// TIA Portal V16 export
// export: Created 2023-03-29T11:04:28.031083Z, ExportSetting WithDefaults, DisplayName Totally Integrated Automation Portal, DisplayVersion V16 Update 6, DisplayName TIA Portal Version Control Interface, DisplayVersion V16 Update 2, DisplayName TIA Portal Openness, DisplayVersion V16 Update 6, DisplayName STEP 7 Professional, DisplayVersion V16 Update 6, DisplayName STEP 7 Safety, DisplayVersion V16, DisplayName WinCC Advanced, DisplayVersion V16 Update 6
ORGANIZATION_BLOCK "OB1"   // OB1, LAD, ProgramCycle
TITLE = Głowny blok
{ S7_Optimized_Access := 'TRUE' }
AUTHOR : RTecmer
VERSION : 0.1
// stored: AutoNumber true, IsIECCheckEnabled false, SetENOAutomatically false
   VAR_INPUT
      Initial_Call : Bool;   // Initial call of this OB
      Remanence : Bool;   // =True, if remanent data are available
   END_VAR
   VAR_TEMP
      tempWatchDog_HMI : Int;
   END_VAR
   VAR_TEMP   // added for the SCL form of the ladder/FBD networks
      _w1 : Bool;
      _w2 : Bool;
   END_VAR
BEGIN

REGION Network 2: Zegart RTC
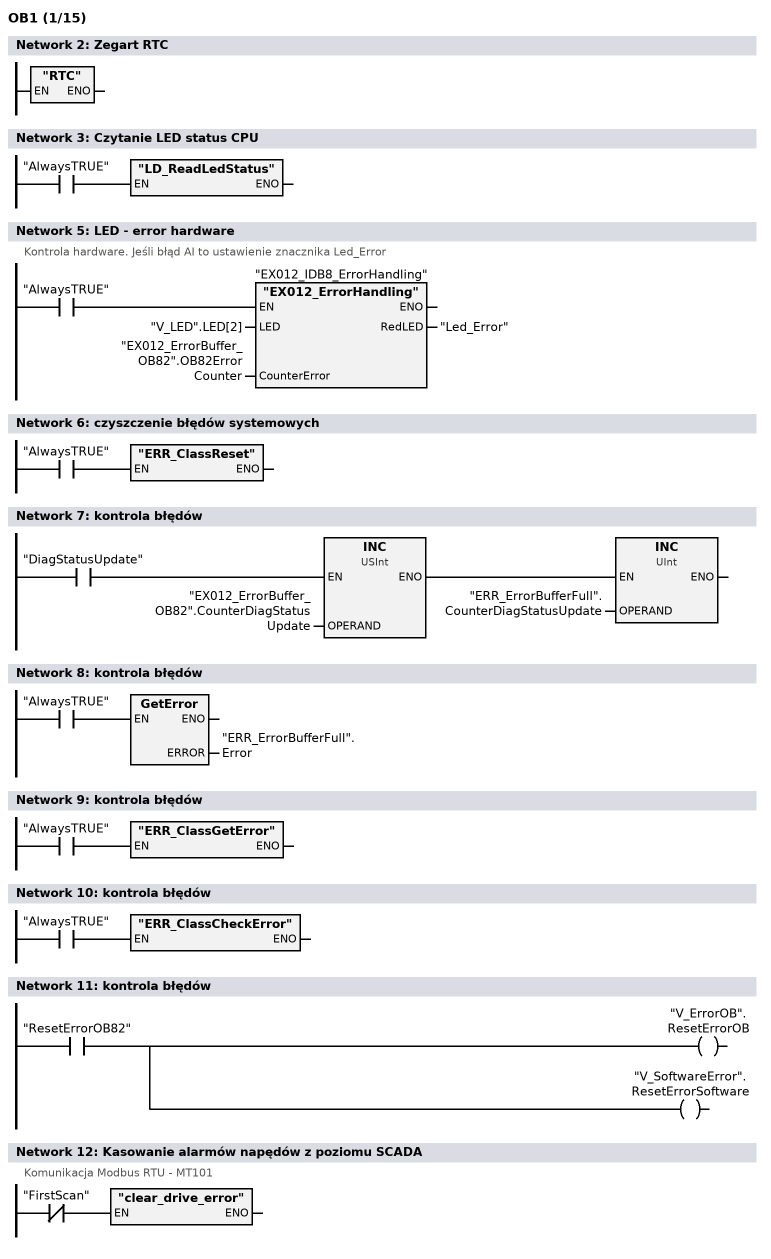
   RUNG wire#powerrail
      "RTC"()
   END_RUNG
   // the same network as SCL:
   "RTC"();
END_REGION

REGION Network 3: Czytanie LED status CPU
   RUNG wire#powerrail
      Contact( "AlwaysTRUE" )
      "LD_ReadLedStatus"()
   END_RUNG
   // the same network as SCL:
   IF "AlwaysTRUE" THEN "LD_ReadLedStatus"(); END_IF;
END_REGION

REGION Network 4 (SCL): LED kontrola RUN
   // Przekazanie  stanu LED 1 CPU
   "DB31_HMI_AreaPointer".getPLCMode := "V_LED".LED[1];
END_REGION

REGION Network 5: LED - error hardware
   // Kontrola hardware. Jeśli błąd AI to ustawienie znacznika Led_Error
   RUNG wire#powerrail
      Contact( "AlwaysTRUE" )
      "EX012_IDB8_ErrorHandling"(LED := "V_LED".LED[2], CounterError := "EX012_ErrorBuffer_OB82".OB82ErrorCounter, RedLED => "Led_Error")
   END_RUNG
   // the same network as SCL:
   IF "AlwaysTRUE" THEN
       "EX012_IDB8_ErrorHandling"(LED := "V_LED".LED[2],   // "EX012_ErrorHandling"
                               CounterError := "EX012_ErrorBuffer_OB82".OB82ErrorCounter,
                               RedLED => "Led_Error");
   END_IF;
END_REGION

REGION Network 6: czyszczenie błędów systemowych
   RUNG wire#powerrail
      Contact( "AlwaysTRUE" )
      "ERR_ClassReset"()
   END_RUNG
   // the same network as SCL:
   IF "AlwaysTRUE" THEN "ERR_ClassReset"(); END_IF;
END_REGION

REGION Network 7: kontrola błędów
   RUNG wire#powerrail
      Contact( "DiagStatusUpdate" )
      { S7_Templates := "DestType := USInt" } Inc( "EX012_ErrorBuffer_OB82".CounterDiagStatusUpdate )
      { S7_Templates := "DestType := UInt" } Inc( "ERR_ErrorBufferFull".CounterDiagStatusUpdate )
   END_RUNG
   // the same network as SCL:
   IF "DiagStatusUpdate" THEN
       "EX012_ErrorBuffer_OB82".CounterDiagStatusUpdate := "EX012_ErrorBuffer_OB82".CounterDiagStatusUpdate + 1;
       "ERR_ErrorBufferFull".CounterDiagStatusUpdate := "ERR_ErrorBufferFull".CounterDiagStatusUpdate + 1;
   END_IF;
END_REGION

REGION Network 8: kontrola błędów
   // no SCL statement known for GetError: written as a call
   IF "AlwaysTRUE" THEN GetError(error => "ERR_ErrorBufferFull".Error); END_IF;
END_REGION

REGION Network 9: kontrola błędów
   RUNG wire#powerrail
      Contact( "AlwaysTRUE" )
      "ERR_ClassGetError"()
   END_RUNG
   // the same network as SCL:
   IF "AlwaysTRUE" THEN "ERR_ClassGetError"(); END_IF;
END_REGION

REGION Network 10: kontrola błędów
   RUNG wire#powerrail
      Contact( "AlwaysTRUE" )
      "ERR_ClassCheckError"()
   END_RUNG
   // the same network as SCL:
   IF "AlwaysTRUE" THEN "ERR_ClassCheckError"(); END_IF;
END_REGION

REGION Network 11: kontrola błędów
   RUNG wire#powerrail
      Contact( "ResetErrorOB82" )
      wire#w1
      Coil( "V_ErrorOB".ResetErrorOB )
   END_RUNG
   RUNG wire#w1
      Coil( "V_SoftwareError".ResetErrorSoftware )
   END_RUNG
   // the same network as SCL:
   "V_ErrorOB".ResetErrorOB := "ResetErrorOB82";
   "V_SoftwareError".ResetErrorSoftware := "ResetErrorOB82";
END_REGION

REGION Network 12: Kasowanie alarmów napędów z poziomu SCADA
   // Komunikacja Modbus RTU - MT101
   RUNG wire#powerrail
      I_Contact( "FirstScan" )
      "clear_drive_error"()
   END_RUNG
   // the same network as SCL:
   IF NOT "FirstScan" THEN "clear_drive_error"(); END_IF;
END_REGION

REGION Network 13: Obsługa przełącznika Tryb Pracy za pośrednictwem SCADA
   // Komunikacja Modbus RTU - MT101
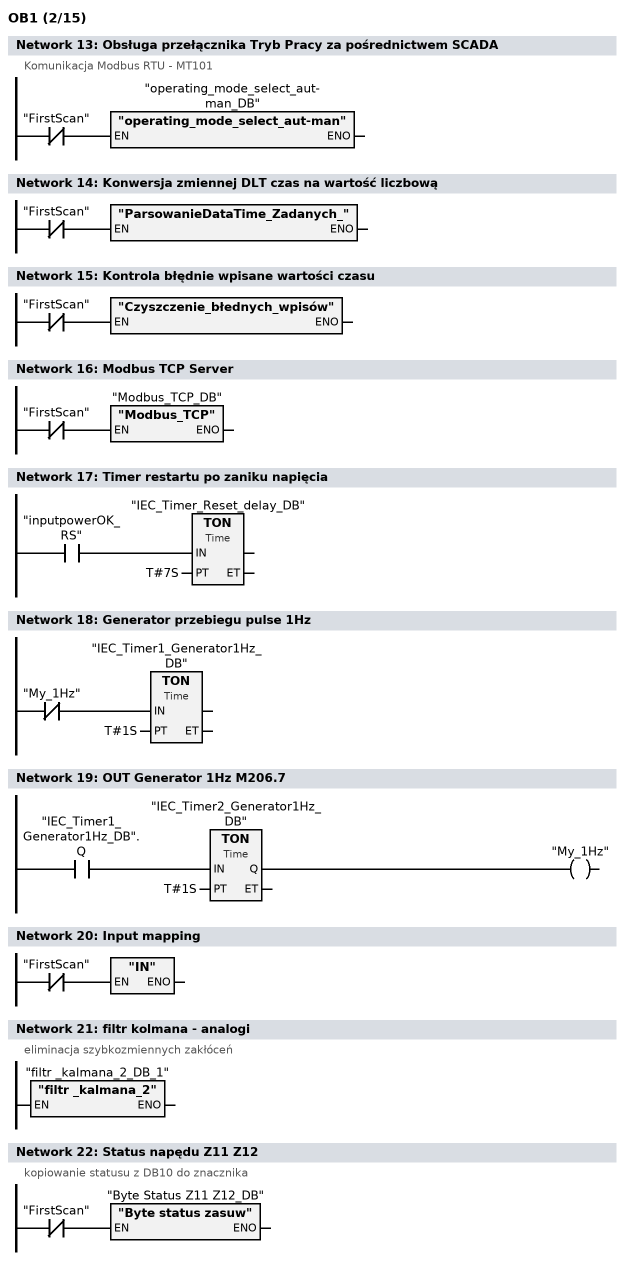
   RUNG wire#powerrail
      I_Contact( "FirstScan" )
      "operating_mode_select_aut-man_DB"()
   END_RUNG
   // the same network as SCL:
   IF NOT "FirstScan" THEN
       "operating_mode_select_aut-man_DB"();   // "operating_mode_select_aut-man"
   END_IF;
END_REGION

REGION Network 14: Konwersja zmiennej DLT czas na wartość liczbową
   RUNG wire#powerrail
      I_Contact( "FirstScan" )
      "ParsowanieDataTime_Zadanych_"()
   END_RUNG
   // the same network as SCL:
   IF NOT "FirstScan" THEN "ParsowanieDataTime_Zadanych_"(); END_IF;
END_REGION

REGION Network 15: Kontrola błędnie wpisane wartości czasu
   RUNG wire#powerrail
      I_Contact( "FirstScan" )
      "Czyszczenie_błednych_wpisów"()
   END_RUNG
   // the same network as SCL:
   IF NOT "FirstScan" THEN "Czyszczenie_błednych_wpisów"(); END_IF;
END_REGION

REGION Network 16: Modbus TCP Server
   RUNG wire#powerrail
      I_Contact( "FirstScan" )
      "Modbus_TCP_DB"()
   END_RUNG
   // the same network as SCL:
   IF NOT "FirstScan" THEN
       "Modbus_TCP_DB"();   // "Modbus_TCP"
   END_IF;
END_REGION

REGION Network 17: Timer restartu po zaniku napięcia
   RUNG wire#powerrail
      Contact( "inputpowerOK_RS" )
      { S7_Templates := "time_type := Time" } "IEC_Timer_Reset_delay_DB".TON(pt := T#7S, et =>)
   END_RUNG
   // the same network as SCL:
   "IEC_Timer_Reset_delay_DB".TON(IN := "inputpowerOK_RS", PT := T#7S);
END_REGION

REGION Network 18: Generator przebiegu pulse 1Hz
   RUNG wire#powerrail
      I_Contact( "My_1Hz" )
      { S7_Templates := "time_type := Time" } "IEC_Timer1_Generator1Hz_DB".TON(pt := T#1S, et =>)
   END_RUNG
   // the same network as SCL:
   "IEC_Timer1_Generator1Hz_DB".TON(IN := NOT "My_1Hz", PT := T#1S);
END_REGION

REGION Network 19: OUT Generator 1Hz M206.7
   RUNG wire#powerrail
      Contact( "IEC_Timer1_Generator1Hz_DB".Q )
      { S7_Templates := "time_type := Time" } "IEC_Timer2_Generator1Hz_DB".TON(pt := T#1S, et =>)
      Coil( "My_1Hz" )
   END_RUNG
   // the same network as SCL:
   "IEC_Timer2_Generator1Hz_DB".TON(IN := "IEC_Timer1_Generator1Hz_DB".Q, PT := T#1S);
   "My_1Hz" := "IEC_Timer2_Generator1Hz_DB".Q;
END_REGION

REGION Network 20: Input mapping
   RUNG wire#powerrail
      I_Contact( "FirstScan" )
      "IN"()
   END_RUNG
   // the same network as SCL:
   IF NOT "FirstScan" THEN "IN"(); END_IF;
END_REGION

REGION Network 21: filtr kolmana - analogi
   // eliminacja szybkozmiennych zakłóceń
   RUNG wire#powerrail
      "filtr _kalmana_2_DB_1"()
   END_RUNG
   // the same network as SCL:
   "filtr _kalmana_2_DB_1"();   // "filtr _kalmana_2"
END_REGION

REGION Network 22: Status napędu Z11 Z12
   // kopiowanie statusu z DB10 do znacznika
   RUNG wire#powerrail
      I_Contact( "FirstScan" )
      "Byte Status Z11 Z12_DB"()
   END_RUNG
   // the same network as SCL:
   IF NOT "FirstScan" THEN
       "Byte Status Z11 Z12_DB"();   // "Byte status zasuw"
   END_IF;
END_REGION

REGION Network 23: RTC HMI - PLC
   // Synchronizacja czasu HMI - PLC
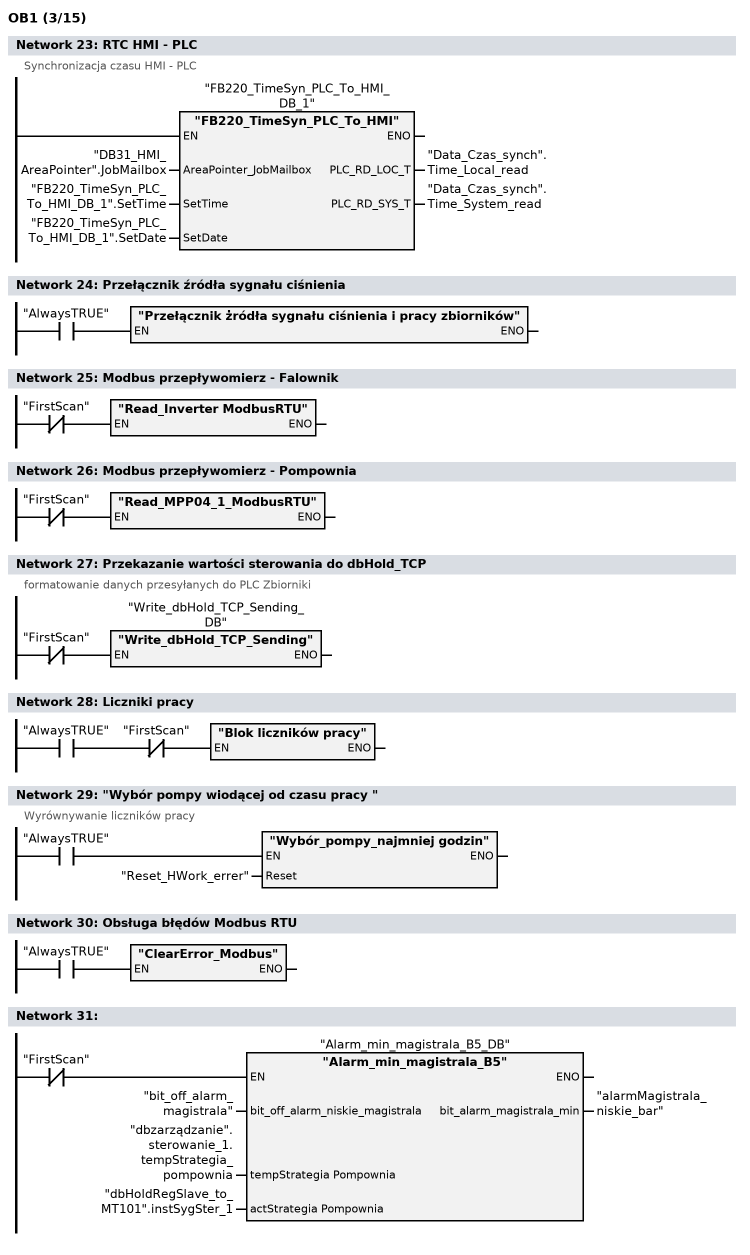
   RUNG wire#powerrail
      "FB220_TimeSyn_PLC_To_HMI_DB_1"(AreaPointer_JobMailbox := "DB31_HMI_AreaPointer".JobMailbox, SetTime := "FB220_TimeSyn_PLC_To_HMI_DB_1".SetTime, SetDate := "FB220_TimeSyn_PLC_To_HMI_DB_1".SetDate, PLC_RD_LOC_T => "Data_Czas_synch".Time_Local_read, PLC_RD_SYS_T => "Data_Czas_synch".Time_System_read)
   END_RUNG
   // the same network as SCL:
   "FB220_TimeSyn_PLC_To_HMI_DB_1"(AreaPointer_JobMailbox := "DB31_HMI_AreaPointer".JobMailbox,   // "FB220_TimeSyn_PLC_To_HMI"
                           SetTime := "FB220_TimeSyn_PLC_To_HMI_DB_1".SetTime,
                           SetDate := "FB220_TimeSyn_PLC_To_HMI_DB_1".SetDate,
                           PLC_RD_LOC_T => "Data_Czas_synch".Time_Local_read,
                           PLC_RD_SYS_T => "Data_Czas_synch".Time_System_read);
END_REGION

REGION Network 24: Przełącznik źródła sygnału ciśnienia
   RUNG wire#powerrail
      Contact( "AlwaysTRUE" )
      "Przełącznik żródła sygnału ciśnienia i pracy zbiorników"()
   END_RUNG
   // the same network as SCL:
   IF "AlwaysTRUE" THEN "Przełącznik żródła sygnału ciśnienia i pracy zbiorników"(); END_IF;
END_REGION

REGION Network 25: Modbus przepływomierz - Falownik
   RUNG wire#powerrail
      I_Contact( "FirstScan" )
      "Read_Inverter ModbusRTU"()
   END_RUNG
   // the same network as SCL:
   IF NOT "FirstScan" THEN "Read_Inverter ModbusRTU"(); END_IF;
END_REGION

REGION Network 26: Modbus przepływomierz - Pompownia
   RUNG wire#powerrail
      I_Contact( "FirstScan" )
      "Read_MPP04_1_ModbusRTU"()
   END_RUNG
   // the same network as SCL:
   IF NOT "FirstScan" THEN "Read_MPP04_1_ModbusRTU"(); END_IF;
END_REGION

REGION Network 27: Przekazanie wartości sterowania do dbHold_TCP
   // formatowanie danych przesyłanych do PLC Zbiorniki
   RUNG wire#powerrail
      I_Contact( "FirstScan" )
      "Write_dbHold_TCP_Sending_DB"()
   END_RUNG
   // the same network as SCL:
   IF NOT "FirstScan" THEN
       "Write_dbHold_TCP_Sending_DB"();   // "Write_dbHold_TCP_Sending"
   END_IF;
END_REGION

REGION Network 28: Liczniki pracy
   RUNG wire#powerrail
      Contact( "AlwaysTRUE" )
      I_Contact( "FirstScan" )
      "Blok liczników pracy"()
   END_RUNG
   // the same network as SCL:
   IF "AlwaysTRUE" AND NOT "FirstScan" THEN "Blok liczników pracy"(); END_IF;
END_REGION

REGION Network 29: "Wybór pompy wiodącej od czasu pracy "
   // Wyrównywanie liczników pracy
   RUNG wire#powerrail
      Contact( "AlwaysTRUE" )
      "Wybór_pompy_najmniej godzin"(Reset := "Reset_HWork_errer")
   END_RUNG
   // the same network as SCL:
   IF "AlwaysTRUE" THEN "Wybór_pompy_najmniej godzin"(Reset := "Reset_HWork_errer"); END_IF;
END_REGION

REGION Network 30: Obsługa błędów Modbus RTU
   RUNG wire#powerrail
      Contact( "AlwaysTRUE" )
      "ClearError_Modbus"()
   END_RUNG
   // the same network as SCL:
   IF "AlwaysTRUE" THEN "ClearError_Modbus"(); END_IF;
END_REGION

REGION Network 31
   RUNG wire#powerrail
      I_Contact( "FirstScan" )
      "Alarm_min_magistrala_B5_DB"(bit_off_alarm_niskie_magistrala := "bit_off_alarm_magistrala", "tempStrategia Pompownia" := "dbzarządzanie".sterowanie_1.tempStrategia_pompownia, "actStrategia Pompownia" := "dbHoldRegSlave_to_MT101".instSygSter_1, bit_alarm_magistrala_min => "alarmMagistrala_niskie_bar")
   END_RUNG
   // the same network as SCL:
   IF NOT "FirstScan" THEN
       "Alarm_min_magistrala_B5_DB"(bit_off_alarm_niskie_magistrala := "bit_off_alarm_magistrala",   // "Alarm_min_magistrala_B5"
                               "tempStrategia Pompownia" := "dbzarządzanie".sterowanie_1.tempStrategia_pompownia,
                               "actStrategia Pompownia" := "dbHoldRegSlave_to_MT101".instSygSter_1,
                               bit_alarm_magistrala_min => "alarmMagistrala_niskie_bar");
   END_IF;
END_REGION

REGION Network 32: Strategia sterowania zasuwami Z11
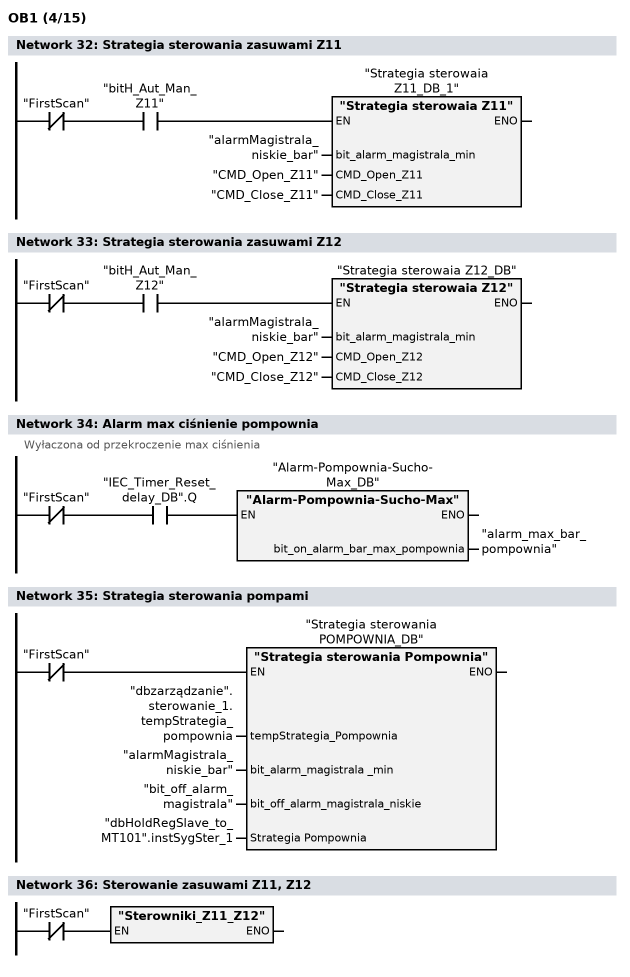
   RUNG wire#powerrail
      I_Contact( "FirstScan" )
      Contact( "bitH_Aut_Man_Z11" )
      "Strategia sterowaia Z11_DB_1"(bit_alarm_magistrala_min := "alarmMagistrala_niskie_bar", CMD_Open_Z11 := "CMD_Open_Z11", CMD_Close_Z11 := "CMD_Close_Z11")
   END_RUNG
   // the same network as SCL:
   IF NOT "FirstScan" AND "bitH_Aut_Man_Z11" THEN
       "Strategia sterowaia Z11_DB_1"(bit_alarm_magistrala_min := "alarmMagistrala_niskie_bar",   // "Strategia sterowaia Z11"
                               CMD_Open_Z11 := "CMD_Open_Z11",
                               CMD_Close_Z11 := "CMD_Close_Z11");
   END_IF;
END_REGION

REGION Network 33: Strategia sterowania zasuwami Z12
   RUNG wire#powerrail
      I_Contact( "FirstScan" )
      Contact( "bitH_Aut_Man_Z12" )
      "Strategia sterowaia Z12_DB"(bit_alarm_magistrala_min := "alarmMagistrala_niskie_bar", CMD_Open_Z12 := "CMD_Open_Z12", CMD_Close_Z12 := "CMD_Close_Z12")
   END_RUNG
   // the same network as SCL:
   IF NOT "FirstScan" AND "bitH_Aut_Man_Z12" THEN
       "Strategia sterowaia Z12_DB"(bit_alarm_magistrala_min := "alarmMagistrala_niskie_bar",   // "Strategia sterowaia Z12"
                               CMD_Open_Z12 := "CMD_Open_Z12",
                               CMD_Close_Z12 := "CMD_Close_Z12");
   END_IF;
END_REGION

REGION Network 34: Alarm max ciśnienie pompownia
   // Wyłaczona od przekroczenie max ciśnienia
   RUNG wire#powerrail
      I_Contact( "FirstScan" )
      Contact( "IEC_Timer_Reset_delay_DB".Q )
      "Alarm-Pompownia-Sucho-Max_DB"(bit_on_alarm_bar_max_pompownia => "alarm_max_bar_pompownia")
   END_RUNG
   // the same network as SCL:
   IF NOT "FirstScan" AND "IEC_Timer_Reset_delay_DB".Q THEN
       "Alarm-Pompownia-Sucho-Max_DB"(bit_on_alarm_bar_max_pompownia => "alarm_max_bar_pompownia");   // "Alarm-Pompownia-Sucho-Max"
   END_IF;
END_REGION

REGION Network 35: Strategia sterowania pompami
   RUNG wire#powerrail
      I_Contact( "FirstScan" )
      "Strategia sterowania POMPOWNIA_DB"(tempStrategia_Pompownia := "dbzarządzanie".sterowanie_1.tempStrategia_pompownia, "bit_alarm_magistrala _min" := "alarmMagistrala_niskie_bar", bit_off_alarm_magistrala_niskie := "bit_off_alarm_magistrala", "Strategia Pompownia" := "dbHoldRegSlave_to_MT101".instSygSter_1)
   END_RUNG
   // the same network as SCL:
   IF NOT "FirstScan" THEN
       "Strategia sterowania POMPOWNIA_DB"(tempStrategia_Pompownia := "dbzarządzanie".sterowanie_1.tempStrategia_pompownia,   // "Strategia sterowania Pompownia"
                               "bit_alarm_magistrala _min" := "alarmMagistrala_niskie_bar",
                               bit_off_alarm_magistrala_niskie := "bit_off_alarm_magistrala",
                               "Strategia Pompownia" := "dbHoldRegSlave_to_MT101".instSygSter_1);
   END_IF;
END_REGION

REGION Network 36: Sterowanie zasuwami Z11, Z12
   RUNG wire#powerrail
      I_Contact( "FirstScan" )
      "Sterowniki_Z11_Z12"()
   END_RUNG
   // the same network as SCL:
   IF NOT "FirstScan" THEN "Sterowniki_Z11_Z12"(); END_IF;
END_REGION

REGION Network 37: Konwerter parametrów z falownika
   // funkcja wylicza wartości pobrane z falownika protokołem Modbus RTU
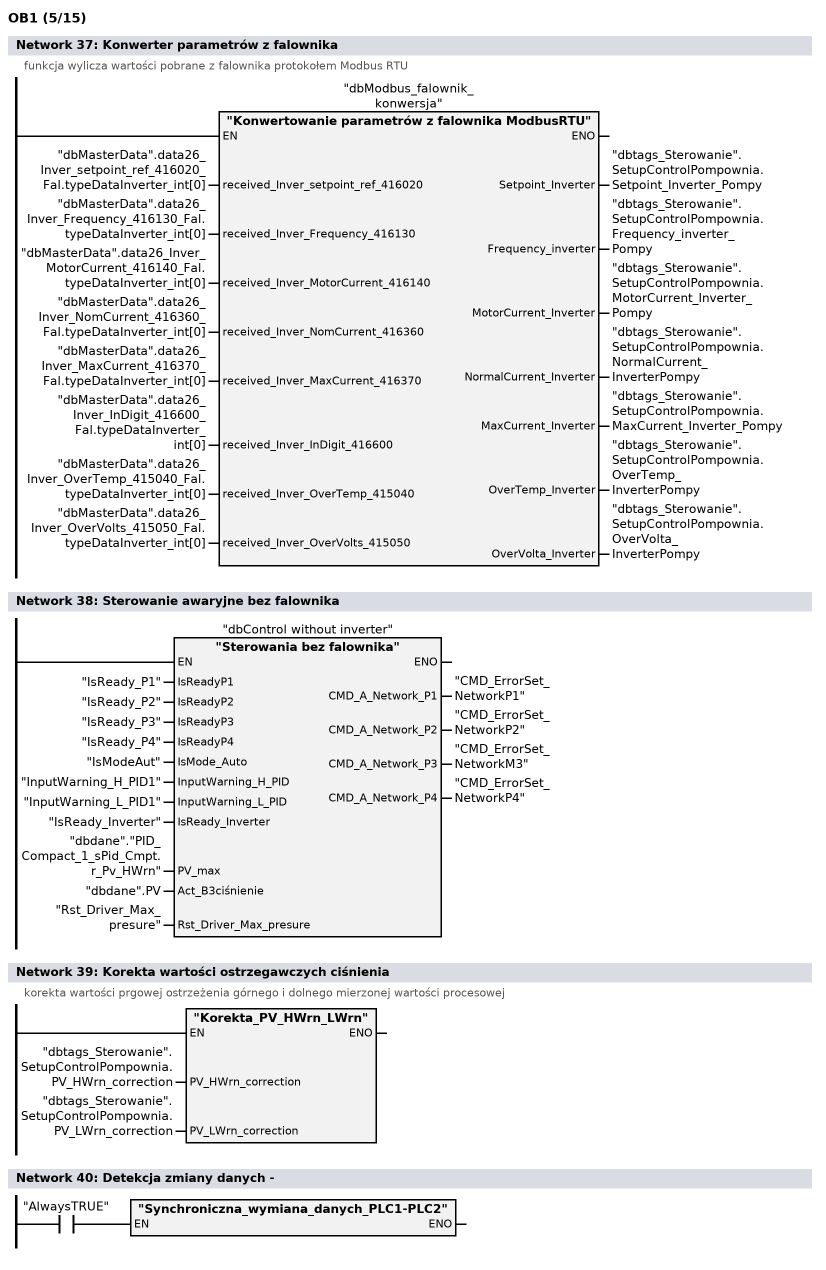
   RUNG wire#powerrail
      "dbModbus_falownik_konwersja"(received_Inver_setpoint_ref_416020 := "dbMasterData".data26_Inver_setpoint_ref_416020_Fal.typeDataInverter_int[0], received_Inver_Frequency_416130 := "dbMasterData".data26_Inver_Frequency_416130_Fal.typeDataInverter_int[0], received_Inver_MotorCurrent_416140 := "dbMasterData".data26_Inver_MotorCurrent_416140_Fal.typeDataInverter_int[0], received_Inver_NomCurrent_416360 := "dbMasterData".data26_Inver_NomCurrent_416360_Fal.typeDataInverter_int[0], received_Inver_MaxCurrent_416370 := "dbMasterData".data26_Inver_MaxCurrent_416370_Fal.typeDataInverter_int[0], received_Inver_InDigit_416600 := "dbMasterData".data26_Inver_InDigit_416600_Fal.typeDataInverter_int[0], received_Inver_OverTemp_415040 := "dbMasterData".data26_Inver_OverTemp_415040_Fal.typeDataInverter_int[0], received_Inver_OverVolts_415050 := "dbMasterData".data26_Inver_OverVolts_415050_Fal.typeDataInverter_int[0], Setpoint_Inverter => "dbtags_Sterowanie".SetupControlPompownia.Setpoint_Inverter_Pompy, Frequency_inverter => "dbtags_Sterowanie".SetupControlPompownia.Frequency_inverter_Pompy, MotorCurrent_Inverter => "dbtags_Sterowanie".SetupControlPompownia.MotorCurrent_Inverter_Pompy, NormalCurrent_Inverter => "dbtags_Sterowanie".SetupControlPompownia.NormalCurrent_InverterPompy, MaxCurrent_Inverter => "dbtags_Sterowanie".SetupControlPompownia.MaxCurrent_Inverter_Pompy, OverTemp_Inverter => "dbtags_Sterowanie".SetupControlPompownia.OverTemp_InverterPompy, OverVolta_Inverter => "dbtags_Sterowanie".SetupControlPompownia.OverVolta_InverterPompy)
   END_RUNG
   // the same network as SCL:
   "dbModbus_falownik_konwersja"(received_Inver_setpoint_ref_416020 := "dbMasterData".data26_Inver_setpoint_ref_416020_Fal.typeDataInverter_int[0],   // "Konwertowanie parametrów z falownika ModbusRTU"
                           received_Inver_Frequency_416130 := "dbMasterData".data26_Inver_Frequency_416130_Fal.typeDataInverter_int[0],
                           received_Inver_MotorCurrent_416140 := "dbMasterData".data26_Inver_MotorCurrent_416140_Fal.typeDataInverter_int[0],
                           received_Inver_NomCurrent_416360 := "dbMasterData".data26_Inver_NomCurrent_416360_Fal.typeDataInverter_int[0],
                           received_Inver_MaxCurrent_416370 := "dbMasterData".data26_Inver_MaxCurrent_416370_Fal.typeDataInverter_int[0],
                           received_Inver_InDigit_416600 := "dbMasterData".data26_Inver_InDigit_416600_Fal.typeDataInverter_int[0],
                           received_Inver_OverTemp_415040 := "dbMasterData".data26_Inver_OverTemp_415040_Fal.typeDataInverter_int[0],
                           received_Inver_OverVolts_415050 := "dbMasterData".data26_Inver_OverVolts_415050_Fal.typeDataInverter_int[0],
                           Setpoint_Inverter => "dbtags_Sterowanie".SetupControlPompownia.Setpoint_Inverter_Pompy,
                           Frequency_inverter => "dbtags_Sterowanie".SetupControlPompownia.Frequency_inverter_Pompy,
                           MotorCurrent_Inverter => "dbtags_Sterowanie".SetupControlPompownia.MotorCurrent_Inverter_Pompy,
                           NormalCurrent_Inverter => "dbtags_Sterowanie".SetupControlPompownia.NormalCurrent_InverterPompy,
                           MaxCurrent_Inverter => "dbtags_Sterowanie".SetupControlPompownia.MaxCurrent_Inverter_Pompy,
                           OverTemp_Inverter => "dbtags_Sterowanie".SetupControlPompownia.OverTemp_InverterPompy,
                           OverVolta_Inverter => "dbtags_Sterowanie".SetupControlPompownia.OverVolta_InverterPompy);
END_REGION

REGION Network 38: Sterowanie awaryjne bez falownika
   RUNG wire#powerrail
      "dbControl without inverter"(IsReadyP1 := "IsReady_P1", IsReadyP2 := "IsReady_P2", IsReadyP3 := "IsReady_P3", IsReadyP4 := "IsReady_P4", IsMode_Auto := "IsModeAut", InputWarning_H_PID := "InputWarning_H_PID1", InputWarning_L_PID := "InputWarning_L_PID1", IsReady_Inverter := "IsReady_Inverter", PV_max := "dbdane"."PID_Compact_1_sPid_Cmpt.r_Pv_HWrn", Act_B3ciśnienie := "dbdane".PV, Rst_Driver_Max_presure := "Rst_Driver_Max_presure", CMD_A_Network_P1 => "CMD_ErrorSet_NetworkP1", CMD_A_Network_P2 => "CMD_ErrorSet_NetworkP2", CMD_A_Network_P3 => "CMD_ErrorSet_NetworkM3", CMD_A_Network_P4 => "CMD_ErrorSet_NetworkP4")
   END_RUNG
   // the same network as SCL:
   "dbControl without inverter"(IsReadyP1 := "IsReady_P1",   // "Sterowania bez falownika"
                           IsReadyP2 := "IsReady_P2",
                           IsReadyP3 := "IsReady_P3",
                           IsReadyP4 := "IsReady_P4",
                           IsMode_Auto := "IsModeAut",
                           InputWarning_H_PID := "InputWarning_H_PID1",
                           InputWarning_L_PID := "InputWarning_L_PID1",
                           IsReady_Inverter := "IsReady_Inverter",
                           PV_max := "dbdane"."PID_Compact_1_sPid_Cmpt.r_Pv_HWrn",
                           Act_B3ciśnienie := "dbdane".PV,
                           Rst_Driver_Max_presure := "Rst_Driver_Max_presure",
                           CMD_A_Network_P1 => "CMD_ErrorSet_NetworkP1",
                           CMD_A_Network_P2 => "CMD_ErrorSet_NetworkP2",
                           CMD_A_Network_P3 => "CMD_ErrorSet_NetworkM3",
                           CMD_A_Network_P4 => "CMD_ErrorSet_NetworkP4");
END_REGION

REGION Network 39: Korekta wartości ostrzegawczych ciśnienia
   // korekta wartości prgowej ostrzeżenia górnego i dolnego mierzonej wartości procesowej
   RUNG wire#powerrail
      "Korekta_PV_HWrn_LWrn"(PV_HWrn_correction := "dbtags_Sterowanie".SetupControlPompownia.PV_HWrn_correction, PV_LWrn_correction := "dbtags_Sterowanie".SetupControlPompownia.PV_LWrn_correction)
   END_RUNG
   // the same network as SCL:
   "Korekta_PV_HWrn_LWrn"(PV_HWrn_correction := "dbtags_Sterowanie".SetupControlPompownia.PV_HWrn_correction,
                          PV_LWrn_correction := "dbtags_Sterowanie".SetupControlPompownia.PV_LWrn_correction);
END_REGION

REGION Network 40: Detekcja zmiany danych -
   RUNG wire#powerrail
      Contact( "AlwaysTRUE" )
      "Synchroniczna_wymiana_danych_PLC1-PLC2"()
   END_RUNG
   // the same network as SCL:
   IF "AlwaysTRUE" THEN "Synchroniczna_wymiana_danych_PLC1-PLC2"(); END_IF;
END_REGION

REGION Network 42: Sterowanie napędami pomp
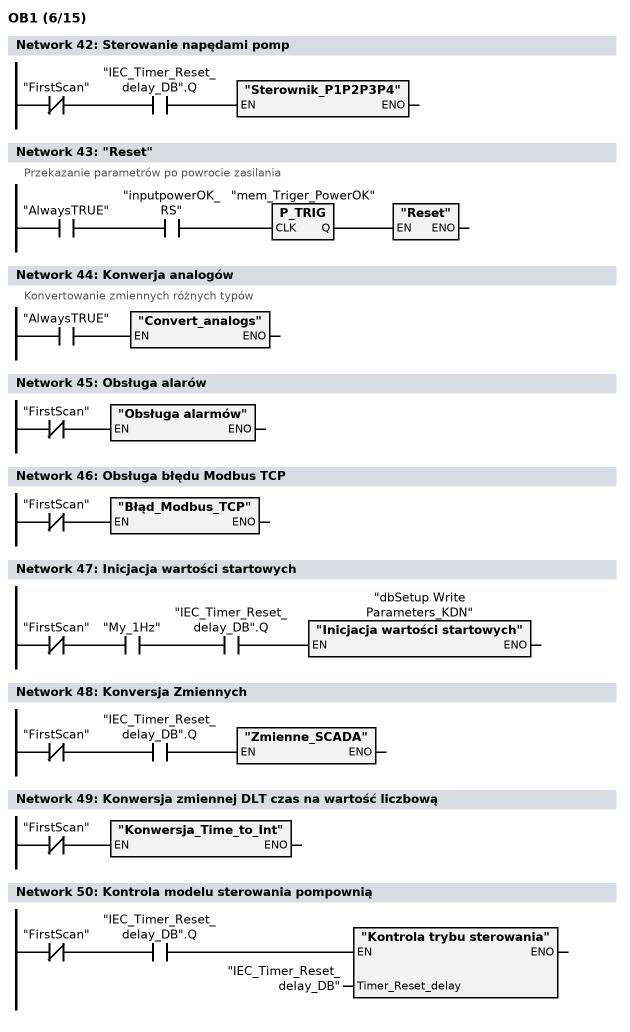
   RUNG wire#powerrail
      I_Contact( "FirstScan" )
      Contact( "IEC_Timer_Reset_delay_DB".Q )
      "Sterownik_P1P2P3P4"()
   END_RUNG
   // the same network as SCL:
   IF NOT "FirstScan" AND "IEC_Timer_Reset_delay_DB".Q THEN "Sterownik_P1P2P3P4"(); END_IF;
END_REGION

REGION Network 43: "Reset"
   // Przekazanie parametrów po powrocie zasilania
   RUNG wire#powerrail
      Contact( "AlwaysTRUE" )
      Contact( "inputpowerOK_RS" )
      P_Trig( "mem_Triger_PowerOK" )
      "Reset"()
   END_RUNG
   // the same network as SCL:
   #_w1 := "AlwaysTRUE" AND "inputpowerOK_RS";
   #_w2 := #_w1 AND NOT "mem_Triger_PowerOK";   // rising edge
   "mem_Triger_PowerOK" := #_w1;
   IF #_w2 THEN "Reset"(); END_IF;
END_REGION

REGION Network 44: Konwerja analogów
   // Konvertowanie zmiennych różnych typów
   RUNG wire#powerrail
      Contact( "AlwaysTRUE" )
      "Convert_analogs"()
   END_RUNG
   // the same network as SCL:
   IF "AlwaysTRUE" THEN "Convert_analogs"(); END_IF;
END_REGION

REGION Network 45: Obsługa alarów
   RUNG wire#powerrail
      I_Contact( "FirstScan" )
      "Obsługa alarmów"()
   END_RUNG
   // the same network as SCL:
   IF NOT "FirstScan" THEN "Obsługa alarmów"(); END_IF;
END_REGION

REGION Network 46: Obsługa błędu Modbus TCP
   RUNG wire#powerrail
      I_Contact( "FirstScan" )
      "Błąd_Modbus_TCP"()
   END_RUNG
   // the same network as SCL:
   IF NOT "FirstScan" THEN "Błąd_Modbus_TCP"(); END_IF;
END_REGION

REGION Network 47: Inicjacja wartości startowych
   RUNG wire#powerrail
      I_Contact( "FirstScan" )
      Contact( "My_1Hz" )
      Contact( "IEC_Timer_Reset_delay_DB".Q )
      "dbSetup Write Parameters_KDN"()
   END_RUNG
   // the same network as SCL:
   IF NOT "FirstScan" AND "My_1Hz" AND "IEC_Timer_Reset_delay_DB".Q THEN
       "dbSetup Write Parameters_KDN"();   // "Inicjacja wartości startowych"
   END_IF;
END_REGION

REGION Network 48: Konversja Zmiennych
   RUNG wire#powerrail
      I_Contact( "FirstScan" )
      Contact( "IEC_Timer_Reset_delay_DB".Q )
      "Zmienne_SCADA"()
   END_RUNG
   // the same network as SCL:
   IF NOT "FirstScan" AND "IEC_Timer_Reset_delay_DB".Q THEN "Zmienne_SCADA"(); END_IF;
END_REGION

REGION Network 49: Konwersja zmiennej DLT czas na wartość liczbową
   RUNG wire#powerrail
      I_Contact( "FirstScan" )
      "Konwersja_Time_to_Int"()
   END_RUNG
   // the same network as SCL:
   IF NOT "FirstScan" THEN "Konwersja_Time_to_Int"(); END_IF;
END_REGION

REGION Network 50: Kontrola modelu sterowania pompownią
   RUNG wire#powerrail
      I_Contact( "FirstScan" )
      Contact( "IEC_Timer_Reset_delay_DB".Q )
      "Kontrola trybu sterowania"(Timer_Reset_delay := "IEC_Timer_Reset_delay_DB")
   END_RUNG
   // the same network as SCL:
   IF NOT "FirstScan" AND "IEC_Timer_Reset_delay_DB".Q THEN
       "Kontrola trybu sterowania"(Timer_Reset_delay := "IEC_Timer_Reset_delay_DB");
   END_IF;
END_REGION

REGION Network 51: Kontrola przyrostu ciśnienia
   // Funkcja w interwale czsowy sprawdza czy następuje przyrost czy spadekciśnienia
   // Wynik podawany jest do funkcji s"Sterowania dodatkową pompą" (Funkacja sterująca doączeniem pompy  dodatkowej)
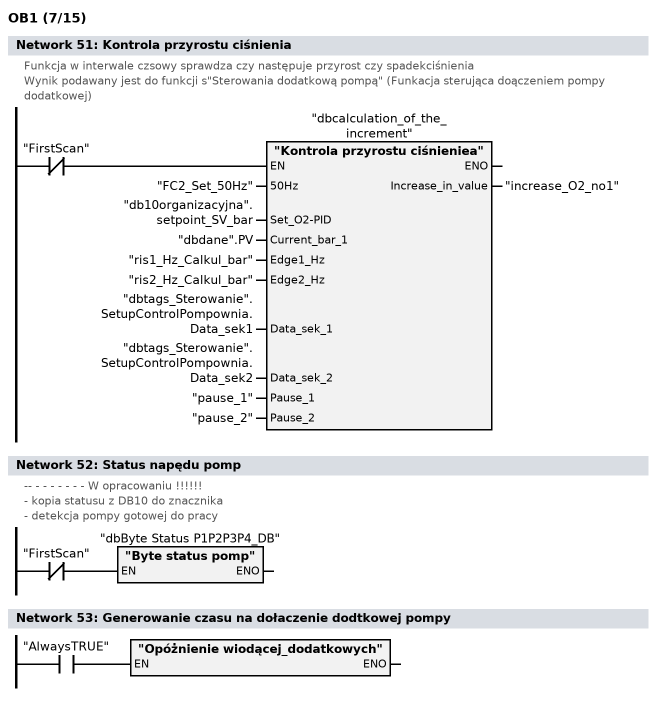
   RUNG wire#powerrail
      I_Contact( "FirstScan" )
      "dbcalculation_of_the_increment"("50Hz" := "FC2_Set_50Hz", "Set_O2-PID" := "db10organizacyjna".setpoint_SV_bar, Current_bar_1 := "dbdane".PV, Edge1_Hz := "ris1_Hz_Calkul_bar", Edge2_Hz := "ris2_Hz_Calkul_bar", Data_sek_1 := "dbtags_Sterowanie".SetupControlPompownia.Data_sek1, Data_sek_2 := "dbtags_Sterowanie".SetupControlPompownia.Data_sek2, Pause_1 := "pause_1", Pause_2 := "pause_2", Increase_in_value => "increase_O2_no1")
   END_RUNG
   // the same network as SCL:
   IF NOT "FirstScan" THEN
       "dbcalculation_of_the_increment"("50Hz" := "FC2_Set_50Hz",   // "Kontrola przyrostu ciśnieniea"
                               "Set_O2-PID" := "db10organizacyjna".setpoint_SV_bar,
                               Current_bar_1 := "dbdane".PV,
                               Edge1_Hz := "ris1_Hz_Calkul_bar",
                               Edge2_Hz := "ris2_Hz_Calkul_bar",
                               Data_sek_1 := "dbtags_Sterowanie".SetupControlPompownia.Data_sek1,
                               Data_sek_2 := "dbtags_Sterowanie".SetupControlPompownia.Data_sek2,
                               Pause_1 := "pause_1",
                               Pause_2 := "pause_2",
                               Increase_in_value => "increase_O2_no1");
   END_IF;
END_REGION

REGION Network 52: Status napędu pomp
   // -- - - - - - - - W opracowaniu !!!!!! 
   // - kopia statusu z DB10 do znacznika
   // - detekcja pompy gotowej do pracy
   RUNG wire#powerrail
      I_Contact( "FirstScan" )
      "dbByte Status P1P2P3P4_DB"()
   END_RUNG
   // the same network as SCL:
   IF NOT "FirstScan" THEN
       "dbByte Status P1P2P3P4_DB"();   // "Byte status pomp"
   END_IF;
END_REGION

REGION Network 53: Generowanie czasu na dołaczenie dodtkowej pompy
   RUNG wire#powerrail
      Contact( "AlwaysTRUE" )
      "Opóżnienie wiodącej_dodatkowych"()
   END_RUNG
   // the same network as SCL:
   IF "AlwaysTRUE" THEN "Opóżnienie wiodącej_dodatkowych"(); END_IF;
END_REGION

REGION Network 54: Sterowanie dołączeniem dodatkowych pomp
   // "dbdane".OUT_PURE_Real
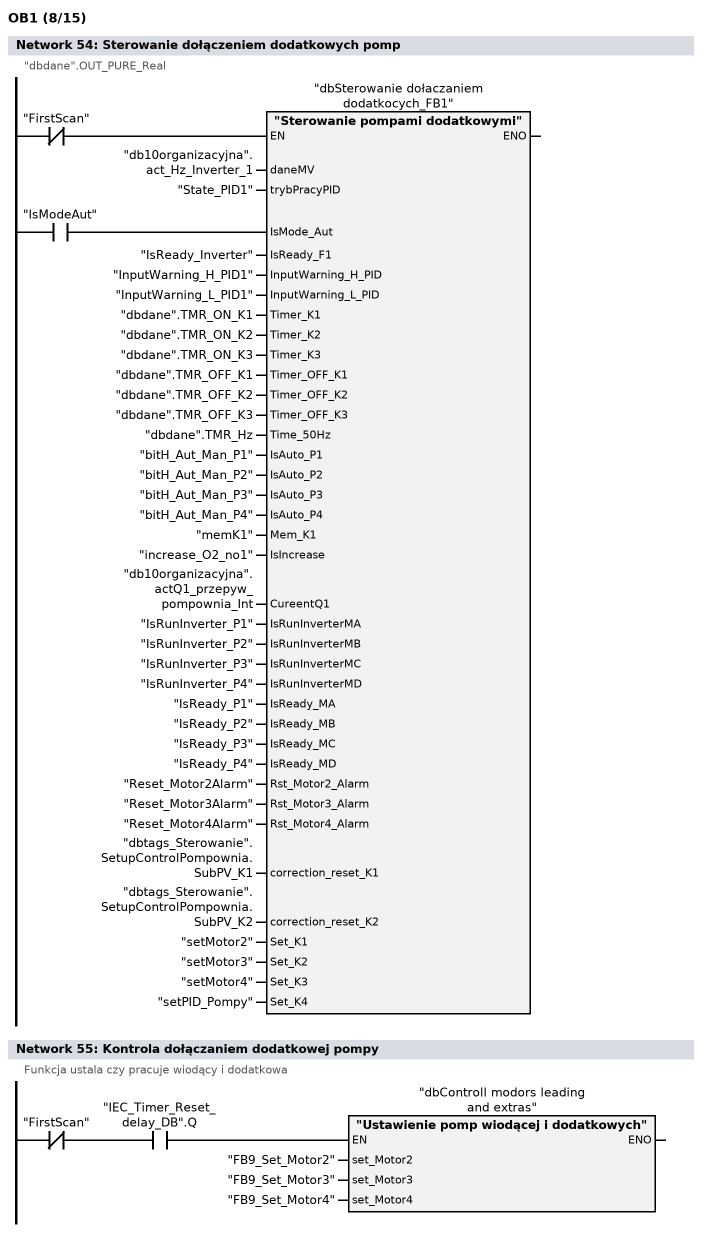
   RUNG wire#powerrail
      I_Contact( "FirstScan" )
      "dbSterowanie dołaczaniem dodatkocych_FB1"(IsMode_Aut := wire#w1, daneMV := "db10organizacyjna".act_Hz_Inverter_1, trybPracyPID := "State_PID1", IsReady_F1 := "IsReady_Inverter", InputWarning_H_PID := "InputWarning_H_PID1", InputWarning_L_PID := "InputWarning_L_PID1", Timer_K1 := "dbdane".TMR_ON_K1, Timer_K2 := "dbdane".TMR_ON_K2, Timer_K3 := "dbdane".TMR_ON_K3, Timer_OFF_K1 := "dbdane".TMR_OFF_K1, Timer_OFF_K2 := "dbdane".TMR_OFF_K2, Timer_OFF_K3 := "dbdane".TMR_OFF_K3, Time_50Hz := "dbdane".TMR_Hz, IsAuto_P1 := "bitH_Aut_Man_P1", IsAuto_P2 := "bitH_Aut_Man_P2", IsAuto_P3 := "bitH_Aut_Man_P3", IsAuto_P4 := "bitH_Aut_Man_P4", Mem_K1 := "memK1", IsIncrease := "increase_O2_no1", CureentQ1 := "db10organizacyjna".actQ1_przepyw_pompownia_Int, IsRunInverterMA := "IsRunInverter_P1", IsRunInverterMB := "IsRunInverter_P2", IsRunInverterMC := "IsRunInverter_P3", IsRunInverterMD := "IsRunInverter_P4", IsReady_MA := "IsReady_P1", IsReady_MB := "IsReady_P2", IsReady_MC := "IsReady_P3", IsReady_MD := "IsReady_P4", Rst_Motor2_Alarm := "Reset_Motor2Alarm", Rst_Motor3_Alarm := "Reset_Motor3Alarm", Rst_Motor4_Alarm := "Reset_Motor4Alarm", correction_reset_K1 := "dbtags_Sterowanie".SetupControlPompownia.SubPV_K1, correction_reset_K2 := "dbtags_Sterowanie".SetupControlPompownia.SubPV_K2, Set_K1 := "setMotor2", Set_K2 := "setMotor3", Set_K3 := "setMotor4", Set_K4 := "setPID_Pompy")
   END_RUNG
   RUNG wire#powerrail
      Contact( "IsModeAut" )
   END_RUNG wire#w1
   // the same network as SCL:
   IF NOT "FirstScan" THEN
       "dbSterowanie dołaczaniem dodatkocych_FB1"(daneMV := "db10organizacyjna".act_Hz_Inverter_1,   // "Sterowanie pompami dodatkowymi"
                               trybPracyPID := "State_PID1",
                               IsMode_Aut := "IsModeAut",
                               IsReady_F1 := "IsReady_Inverter",
                               InputWarning_H_PID := "InputWarning_H_PID1",
                               InputWarning_L_PID := "InputWarning_L_PID1",
                               Timer_K1 := "dbdane".TMR_ON_K1,
                               Timer_K2 := "dbdane".TMR_ON_K2,
                               Timer_K3 := "dbdane".TMR_ON_K3,
                               Timer_OFF_K1 := "dbdane".TMR_OFF_K1,
                               Timer_OFF_K2 := "dbdane".TMR_OFF_K2,
                               Timer_OFF_K3 := "dbdane".TMR_OFF_K3,
                               Time_50Hz := "dbdane".TMR_Hz,
                               IsAuto_P1 := "bitH_Aut_Man_P1",
                               IsAuto_P2 := "bitH_Aut_Man_P2",
                               IsAuto_P3 := "bitH_Aut_Man_P3",
                               IsAuto_P4 := "bitH_Aut_Man_P4",
                               Mem_K1 := "memK1",
                               IsIncrease := "increase_O2_no1",
                               CureentQ1 := "db10organizacyjna".actQ1_przepyw_pompownia_Int,
                               IsRunInverterMA := "IsRunInverter_P1",
                               IsRunInverterMB := "IsRunInverter_P2",
                               IsRunInverterMC := "IsRunInverter_P3",
                               IsRunInverterMD := "IsRunInverter_P4",
                               IsReady_MA := "IsReady_P1",
                               IsReady_MB := "IsReady_P2",
                               IsReady_MC := "IsReady_P3",
                               IsReady_MD := "IsReady_P4",
                               Rst_Motor2_Alarm := "Reset_Motor2Alarm",
                               Rst_Motor3_Alarm := "Reset_Motor3Alarm",
                               Rst_Motor4_Alarm := "Reset_Motor4Alarm",
                               correction_reset_K1 := "dbtags_Sterowanie".SetupControlPompownia.SubPV_K1,
                               correction_reset_K2 := "dbtags_Sterowanie".SetupControlPompownia.SubPV_K2,
                               Set_K1 := "setMotor2",
                               Set_K2 := "setMotor3",
                               Set_K3 := "setMotor4",
                               Set_K4 := "setPID_Pompy");
   END_IF;
END_REGION

REGION Network 55: Kontrola dołączaniem dodatkowej pompy
   // Funkcja ustala czy pracuje wiodący i dodatkowa
   RUNG wire#powerrail
      I_Contact( "FirstScan" )
      Contact( "IEC_Timer_Reset_delay_DB".Q )
      "dbControll modors leading and extras"(set_Motor2 := "FB9_Set_Motor2", set_Motor3 := "FB9_Set_Motor3", set_Motor4 := "FB9_Set_Motor4")
   END_RUNG
   // the same network as SCL:
   IF NOT "FirstScan" AND "IEC_Timer_Reset_delay_DB".Q THEN
       "dbControll modors leading and extras"(set_Motor2 := "FB9_Set_Motor2",   // "Ustawienie pomp wiodącej i dodatkowych"
                               set_Motor3 := "FB9_Set_Motor3",
                               set_Motor4 := "FB9_Set_Motor4");
   END_IF;
END_REGION

REGION Network 56: Falownik P1
   // Sterowaniem pracy z falownika. Sterowanie napędem na pozycji MC
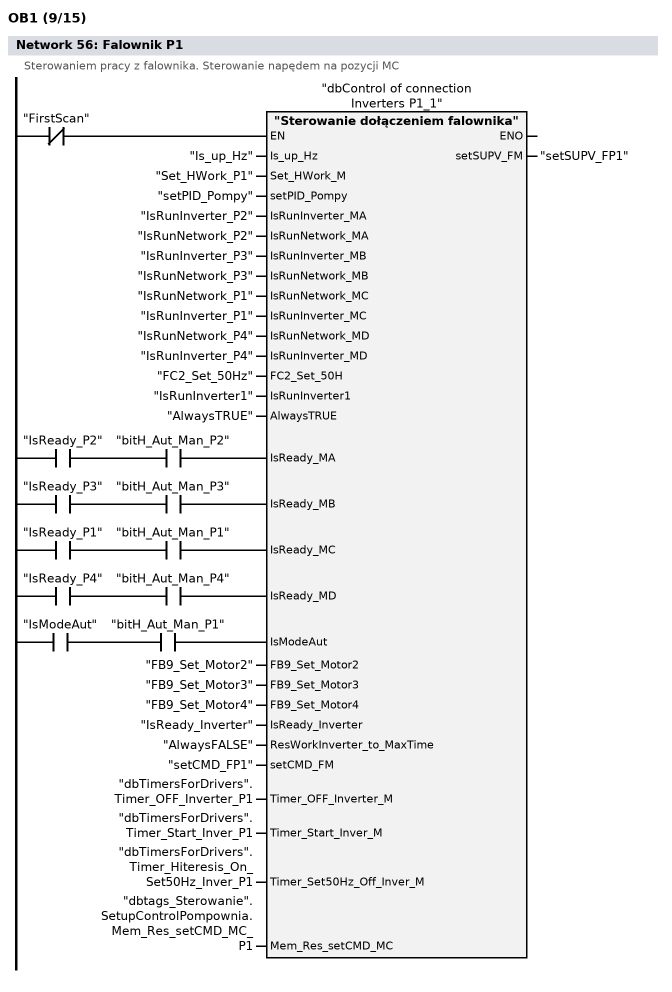
   RUNG wire#powerrail
      I_Contact( "FirstScan" )
      "dbControl of connection Inverters P1_1"(IsReady_MA := wire#w1, IsReady_MB := wire#w2, IsReady_MC := wire#w3, IsReady_MD := wire#w4, IsModeAut := wire#w5, Is_up_Hz := "Is_up_Hz", Set_HWork_M := "Set_HWork_P1", setPID_Pompy := "setPID_Pompy", IsRunInverter_MA := "IsRunInverter_P2", IsRunNetwork_MA := "IsRunNetwork_P2", IsRunInverter_MB := "IsRunInverter_P3", IsRunNetwork_MB := "IsRunNetwork_P3", IsRunNetwork_MC := "IsRunNetwork_P1", IsRunInverter_MC := "IsRunInverter_P1", IsRunNetwork_MD := "IsRunNetwork_P4", IsRunInverter_MD := "IsRunInverter_P4", FC2_Set_50H := "FC2_Set_50Hz", IsRunInverter1 := "IsRunInverter1", AlwaysTRUE := "AlwaysTRUE", FB9_Set_Motor2 := "FB9_Set_Motor2", FB9_Set_Motor3 := "FB9_Set_Motor3", FB9_Set_Motor4 := "FB9_Set_Motor4", IsReady_Inverter := "IsReady_Inverter", ResWorkInverter_to_MaxTime := "AlwaysFALSE", setCMD_FM := "setCMD_FP1", Timer_OFF_Inverter_M := "dbTimersForDrivers".Timer_OFF_Inverter_P1, Timer_Start_Inver_M := "dbTimersForDrivers".Timer_Start_Inver_P1, Timer_Set50Hz_Off_Inver_M := "dbTimersForDrivers".Timer_Hiteresis_On_Set50Hz_Inver_P1, Mem_Res_setCMD_MC := "dbtags_Sterowanie".SetupControlPompownia.Mem_Res_setCMD_MC_P1, setSUPV_FM => "setSUPV_FP1")
   END_RUNG
   RUNG wire#powerrail
      Contact( "IsReady_P2" )
      Contact( "bitH_Aut_Man_P2" )
   END_RUNG wire#w1
   RUNG wire#powerrail
      Contact( "IsReady_P3" )
      Contact( "bitH_Aut_Man_P3" )
   END_RUNG wire#w2
   RUNG wire#powerrail
      Contact( "IsReady_P1" )
      Contact( "bitH_Aut_Man_P1" )
   END_RUNG wire#w3
   RUNG wire#powerrail
      Contact( "IsReady_P4" )
      Contact( "bitH_Aut_Man_P4" )
   END_RUNG wire#w4
   RUNG wire#powerrail
      Contact( "IsModeAut" )
      Contact( "bitH_Aut_Man_P1" )
   END_RUNG wire#w5
   // the same network as SCL:
   IF NOT "FirstScan" THEN
       "dbControl of connection Inverters P1_1"(Is_up_Hz := "Is_up_Hz",   // "Sterowanie dołączeniem falownika"
                               Set_HWork_M := "Set_HWork_P1",
                               setPID_Pompy := "setPID_Pompy",
                               IsRunInverter_MA := "IsRunInverter_P2",
                               IsRunNetwork_MA := "IsRunNetwork_P2",
                               IsRunInverter_MB := "IsRunInverter_P3",
                               IsRunNetwork_MB := "IsRunNetwork_P3",
                               IsRunNetwork_MC := "IsRunNetwork_P1",
                               IsRunInverter_MC := "IsRunInverter_P1",
                               IsRunNetwork_MD := "IsRunNetwork_P4",
                               IsRunInverter_MD := "IsRunInverter_P4",
                               FC2_Set_50H := "FC2_Set_50Hz",
                               IsRunInverter1 := "IsRunInverter1",
                               AlwaysTRUE := "AlwaysTRUE",
                               IsReady_MA := "IsReady_P2" AND "bitH_Aut_Man_P2",
                               IsReady_MB := "IsReady_P3" AND "bitH_Aut_Man_P3",
                               IsReady_MC := "IsReady_P1" AND "bitH_Aut_Man_P1",
                               IsReady_MD := "IsReady_P4" AND "bitH_Aut_Man_P4",
                               IsModeAut := "IsModeAut" AND "bitH_Aut_Man_P1",
                               FB9_Set_Motor2 := "FB9_Set_Motor2",
                               FB9_Set_Motor3 := "FB9_Set_Motor3",
                               FB9_Set_Motor4 := "FB9_Set_Motor4",
                               IsReady_Inverter := "IsReady_Inverter",
                               ResWorkInverter_to_MaxTime := "AlwaysFALSE",
                               setCMD_FM := "setCMD_FP1",
                               Timer_OFF_Inverter_M := "dbTimersForDrivers".Timer_OFF_Inverter_P1,
                               Timer_Start_Inver_M := "dbTimersForDrivers".Timer_Start_Inver_P1,
                               Timer_Set50Hz_Off_Inver_M := "dbTimersForDrivers".Timer_Hiteresis_On_Set50Hz_Inver_P1,
                               Mem_Res_setCMD_MC := "dbtags_Sterowanie".SetupControlPompownia.Mem_Res_setCMD_MC_P1,
                               setSUPV_FM => "setSUPV_FP1");
   END_IF;
END_REGION

REGION Network 57: Falownik P2
   // Sterowaniem pracy z falownika. Sterowanie napędem na pozycji MC
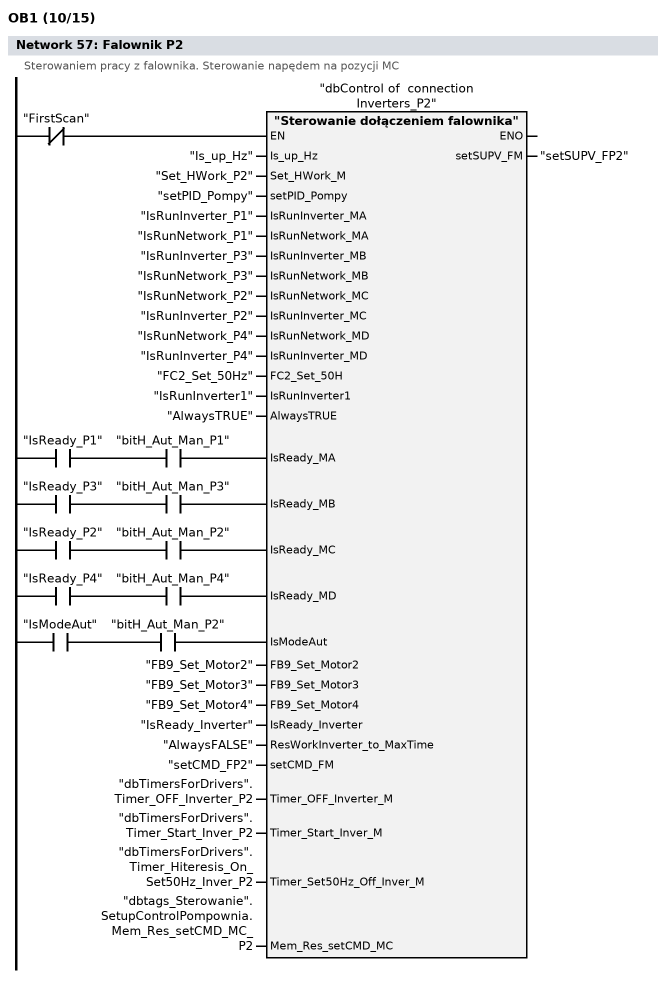
   RUNG wire#powerrail
      I_Contact( "FirstScan" )
      "dbControl of  connection Inverters_P2"(IsReady_MA := wire#w1, IsReady_MB := wire#w2, IsReady_MC := wire#w3, IsReady_MD := wire#w4, IsModeAut := wire#w5, Is_up_Hz := "Is_up_Hz", Set_HWork_M := "Set_HWork_P2", setPID_Pompy := "setPID_Pompy", IsRunInverter_MA := "IsRunInverter_P1", IsRunNetwork_MA := "IsRunNetwork_P1", IsRunInverter_MB := "IsRunInverter_P3", IsRunNetwork_MB := "IsRunNetwork_P3", IsRunNetwork_MC := "IsRunNetwork_P2", IsRunInverter_MC := "IsRunInverter_P2", IsRunNetwork_MD := "IsRunNetwork_P4", IsRunInverter_MD := "IsRunInverter_P4", FC2_Set_50H := "FC2_Set_50Hz", IsRunInverter1 := "IsRunInverter1", AlwaysTRUE := "AlwaysTRUE", FB9_Set_Motor2 := "FB9_Set_Motor2", FB9_Set_Motor3 := "FB9_Set_Motor3", FB9_Set_Motor4 := "FB9_Set_Motor4", IsReady_Inverter := "IsReady_Inverter", ResWorkInverter_to_MaxTime := "AlwaysFALSE", setCMD_FM := "setCMD_FP2", Timer_OFF_Inverter_M := "dbTimersForDrivers".Timer_OFF_Inverter_P2, Timer_Start_Inver_M := "dbTimersForDrivers".Timer_Start_Inver_P2, Timer_Set50Hz_Off_Inver_M := "dbTimersForDrivers".Timer_Hiteresis_On_Set50Hz_Inver_P2, Mem_Res_setCMD_MC := "dbtags_Sterowanie".SetupControlPompownia.Mem_Res_setCMD_MC_P2, setSUPV_FM => "setSUPV_FP2")
   END_RUNG
   RUNG wire#powerrail
      Contact( "IsReady_P1" )
      Contact( "bitH_Aut_Man_P1" )
   END_RUNG wire#w1
   RUNG wire#powerrail
      Contact( "IsReady_P3" )
      Contact( "bitH_Aut_Man_P3" )
   END_RUNG wire#w2
   RUNG wire#powerrail
      Contact( "IsReady_P2" )
      Contact( "bitH_Aut_Man_P2" )
   END_RUNG wire#w3
   RUNG wire#powerrail
      Contact( "IsReady_P4" )
      Contact( "bitH_Aut_Man_P4" )
   END_RUNG wire#w4
   RUNG wire#powerrail
      Contact( "IsModeAut" )
      Contact( "bitH_Aut_Man_P2" )
   END_RUNG wire#w5
   // the same network as SCL:
   IF NOT "FirstScan" THEN
       "dbControl of  connection Inverters_P2"(Is_up_Hz := "Is_up_Hz",   // "Sterowanie dołączeniem falownika"
                               Set_HWork_M := "Set_HWork_P2",
                               setPID_Pompy := "setPID_Pompy",
                               IsRunInverter_MA := "IsRunInverter_P1",
                               IsRunNetwork_MA := "IsRunNetwork_P1",
                               IsRunInverter_MB := "IsRunInverter_P3",
                               IsRunNetwork_MB := "IsRunNetwork_P3",
                               IsRunNetwork_MC := "IsRunNetwork_P2",
                               IsRunInverter_MC := "IsRunInverter_P2",
                               IsRunNetwork_MD := "IsRunNetwork_P4",
                               IsRunInverter_MD := "IsRunInverter_P4",
                               FC2_Set_50H := "FC2_Set_50Hz",
                               IsRunInverter1 := "IsRunInverter1",
                               AlwaysTRUE := "AlwaysTRUE",
                               IsReady_MA := "IsReady_P1" AND "bitH_Aut_Man_P1",
                               IsReady_MB := "IsReady_P3" AND "bitH_Aut_Man_P3",
                               IsReady_MC := "IsReady_P2" AND "bitH_Aut_Man_P2",
                               IsReady_MD := "IsReady_P4" AND "bitH_Aut_Man_P4",
                               IsModeAut := "IsModeAut" AND "bitH_Aut_Man_P2",
                               FB9_Set_Motor2 := "FB9_Set_Motor2",
                               FB9_Set_Motor3 := "FB9_Set_Motor3",
                               FB9_Set_Motor4 := "FB9_Set_Motor4",
                               IsReady_Inverter := "IsReady_Inverter",
                               ResWorkInverter_to_MaxTime := "AlwaysFALSE",
                               setCMD_FM := "setCMD_FP2",
                               Timer_OFF_Inverter_M := "dbTimersForDrivers".Timer_OFF_Inverter_P2,
                               Timer_Start_Inver_M := "dbTimersForDrivers".Timer_Start_Inver_P2,
                               Timer_Set50Hz_Off_Inver_M := "dbTimersForDrivers".Timer_Hiteresis_On_Set50Hz_Inver_P2,
                               Mem_Res_setCMD_MC := "dbtags_Sterowanie".SetupControlPompownia.Mem_Res_setCMD_MC_P2,
                               setSUPV_FM => "setSUPV_FP2");
   END_IF;
END_REGION

REGION Network 58: Falownik P3
   // Sterowaniem pracy z falownika. Sterowanie napędem na pozycji MC
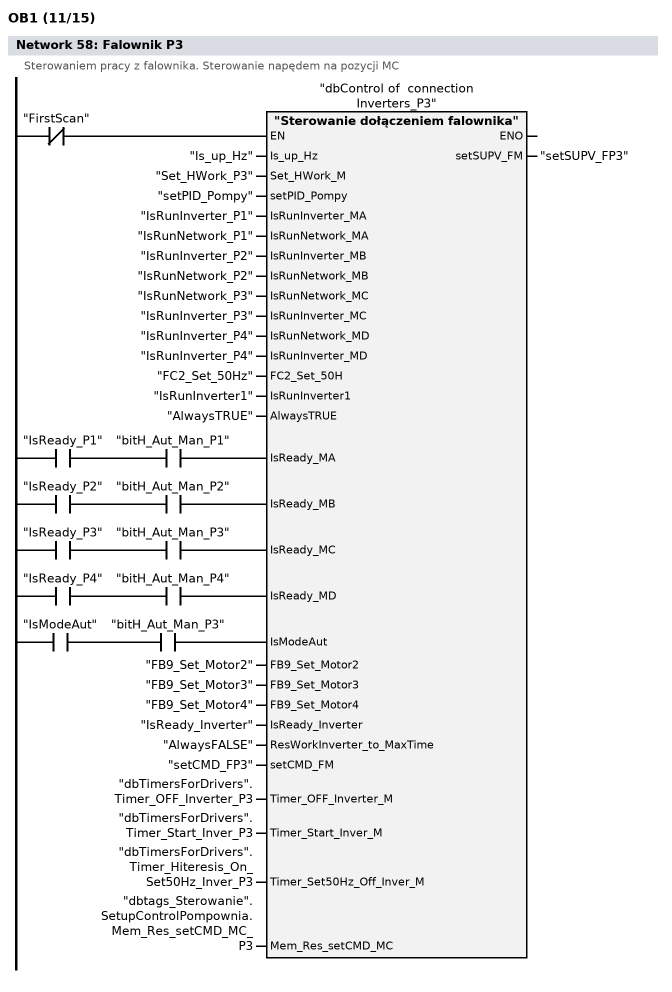
   RUNG wire#powerrail
      I_Contact( "FirstScan" )
      "dbControl of  connection Inverters_P3"(IsReady_MA := wire#w1, IsReady_MB := wire#w2, IsReady_MC := wire#w3, IsReady_MD := wire#w4, IsModeAut := wire#w5, Is_up_Hz := "Is_up_Hz", Set_HWork_M := "Set_HWork_P3", setPID_Pompy := "setPID_Pompy", IsRunInverter_MA := "IsRunInverter_P1", IsRunNetwork_MA := "IsRunNetwork_P1", IsRunInverter_MB := "IsRunInverter_P2", IsRunNetwork_MB := "IsRunNetwork_P2", IsRunNetwork_MC := "IsRunNetwork_P3", IsRunInverter_MC := "IsRunInverter_P3", IsRunNetwork_MD := "IsRunInverter_P4", IsRunInverter_MD := "IsRunInverter_P4", FC2_Set_50H := "FC2_Set_50Hz", IsRunInverter1 := "IsRunInverter1", AlwaysTRUE := "AlwaysTRUE", FB9_Set_Motor2 := "FB9_Set_Motor2", FB9_Set_Motor3 := "FB9_Set_Motor3", FB9_Set_Motor4 := "FB9_Set_Motor4", IsReady_Inverter := "IsReady_Inverter", ResWorkInverter_to_MaxTime := "AlwaysFALSE", setCMD_FM := "setCMD_FP3", Timer_OFF_Inverter_M := "dbTimersForDrivers".Timer_OFF_Inverter_P3, Timer_Start_Inver_M := "dbTimersForDrivers".Timer_Start_Inver_P3, Timer_Set50Hz_Off_Inver_M := "dbTimersForDrivers".Timer_Hiteresis_On_Set50Hz_Inver_P3, Mem_Res_setCMD_MC := "dbtags_Sterowanie".SetupControlPompownia.Mem_Res_setCMD_MC_P3, setSUPV_FM => "setSUPV_FP3")
   END_RUNG
   RUNG wire#powerrail
      Contact( "IsReady_P1" )
      Contact( "bitH_Aut_Man_P1" )
   END_RUNG wire#w1
   RUNG wire#powerrail
      Contact( "IsReady_P2" )
      Contact( "bitH_Aut_Man_P2" )
   END_RUNG wire#w2
   RUNG wire#powerrail
      Contact( "IsReady_P3" )
      Contact( "bitH_Aut_Man_P3" )
   END_RUNG wire#w3
   RUNG wire#powerrail
      Contact( "IsReady_P4" )
      Contact( "bitH_Aut_Man_P4" )
   END_RUNG wire#w4
   RUNG wire#powerrail
      Contact( "IsModeAut" )
      Contact( "bitH_Aut_Man_P3" )
   END_RUNG wire#w5
   // the same network as SCL:
   IF NOT "FirstScan" THEN
       "dbControl of  connection Inverters_P3"(Is_up_Hz := "Is_up_Hz",   // "Sterowanie dołączeniem falownika"
                               Set_HWork_M := "Set_HWork_P3",
                               setPID_Pompy := "setPID_Pompy",
                               IsRunInverter_MA := "IsRunInverter_P1",
                               IsRunNetwork_MA := "IsRunNetwork_P1",
                               IsRunInverter_MB := "IsRunInverter_P2",
                               IsRunNetwork_MB := "IsRunNetwork_P2",
                               IsRunNetwork_MC := "IsRunNetwork_P3",
                               IsRunInverter_MC := "IsRunInverter_P3",
                               IsRunNetwork_MD := "IsRunInverter_P4",
                               IsRunInverter_MD := "IsRunInverter_P4",
                               FC2_Set_50H := "FC2_Set_50Hz",
                               IsRunInverter1 := "IsRunInverter1",
                               AlwaysTRUE := "AlwaysTRUE",
                               IsReady_MA := "IsReady_P1" AND "bitH_Aut_Man_P1",
                               IsReady_MB := "IsReady_P2" AND "bitH_Aut_Man_P2",
                               IsReady_MC := "IsReady_P3" AND "bitH_Aut_Man_P3",
                               IsReady_MD := "IsReady_P4" AND "bitH_Aut_Man_P4",
                               IsModeAut := "IsModeAut" AND "bitH_Aut_Man_P3",
                               FB9_Set_Motor2 := "FB9_Set_Motor2",
                               FB9_Set_Motor3 := "FB9_Set_Motor3",
                               FB9_Set_Motor4 := "FB9_Set_Motor4",
                               IsReady_Inverter := "IsReady_Inverter",
                               ResWorkInverter_to_MaxTime := "AlwaysFALSE",
                               setCMD_FM := "setCMD_FP3",
                               Timer_OFF_Inverter_M := "dbTimersForDrivers".Timer_OFF_Inverter_P3,
                               Timer_Start_Inver_M := "dbTimersForDrivers".Timer_Start_Inver_P3,
                               Timer_Set50Hz_Off_Inver_M := "dbTimersForDrivers".Timer_Hiteresis_On_Set50Hz_Inver_P3,
                               Mem_Res_setCMD_MC := "dbtags_Sterowanie".SetupControlPompownia.Mem_Res_setCMD_MC_P3,
                               setSUPV_FM => "setSUPV_FP3");
   END_IF;
END_REGION

REGION Network 59: Falownik P4
   // Sterowaniem pracy z falownika. Sterowanie napędem na pozycji MC
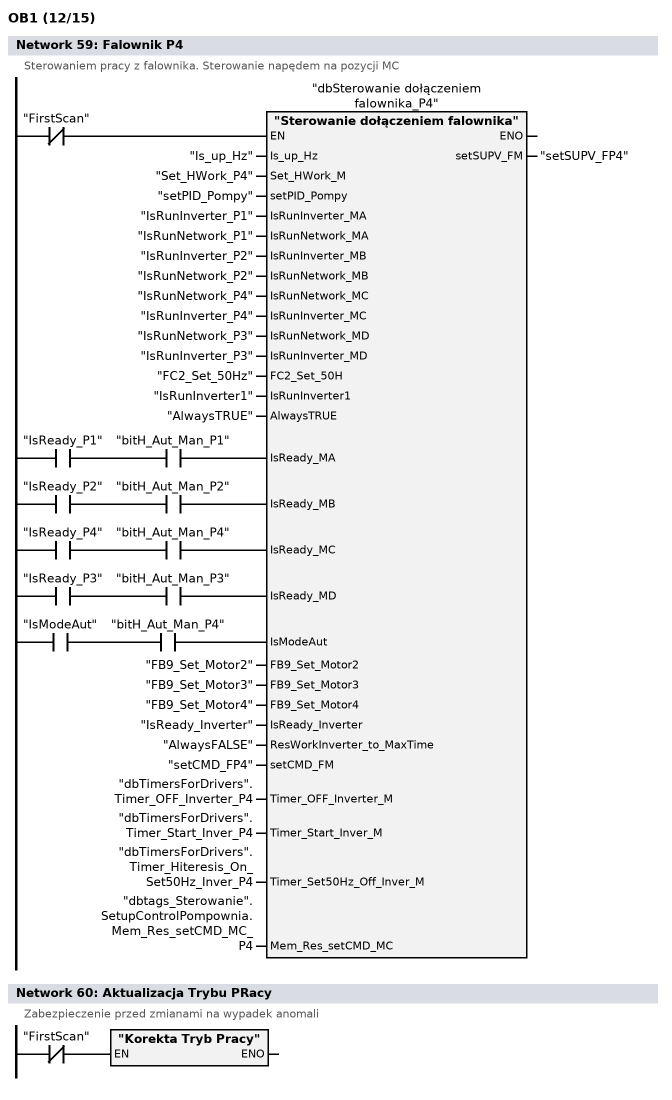
   RUNG wire#powerrail
      I_Contact( "FirstScan" )
      "dbSterowanie dołączeniem falownika_P4"(IsReady_MA := wire#w1, IsReady_MB := wire#w2, IsReady_MC := wire#w3, IsReady_MD := wire#w4, IsModeAut := wire#w5, Is_up_Hz := "Is_up_Hz", Set_HWork_M := "Set_HWork_P4", setPID_Pompy := "setPID_Pompy", IsRunInverter_MA := "IsRunInverter_P1", IsRunNetwork_MA := "IsRunNetwork_P1", IsRunInverter_MB := "IsRunInverter_P2", IsRunNetwork_MB := "IsRunNetwork_P2", IsRunNetwork_MC := "IsRunNetwork_P4", IsRunInverter_MC := "IsRunInverter_P4", IsRunNetwork_MD := "IsRunNetwork_P3", IsRunInverter_MD := "IsRunInverter_P3", FC2_Set_50H := "FC2_Set_50Hz", IsRunInverter1 := "IsRunInverter1", AlwaysTRUE := "AlwaysTRUE", FB9_Set_Motor2 := "FB9_Set_Motor2", FB9_Set_Motor3 := "FB9_Set_Motor3", FB9_Set_Motor4 := "FB9_Set_Motor4", IsReady_Inverter := "IsReady_Inverter", ResWorkInverter_to_MaxTime := "AlwaysFALSE", setCMD_FM := "setCMD_FP4", Timer_OFF_Inverter_M := "dbTimersForDrivers".Timer_OFF_Inverter_P4, Timer_Start_Inver_M := "dbTimersForDrivers".Timer_Start_Inver_P4, Timer_Set50Hz_Off_Inver_M := "dbTimersForDrivers".Timer_Hiteresis_On_Set50Hz_Inver_P4, Mem_Res_setCMD_MC := "dbtags_Sterowanie".SetupControlPompownia.Mem_Res_setCMD_MC_P4, setSUPV_FM => "setSUPV_FP4")
   END_RUNG
   RUNG wire#powerrail
      Contact( "IsReady_P1" )
      Contact( "bitH_Aut_Man_P1" )
   END_RUNG wire#w1
   RUNG wire#powerrail
      Contact( "IsReady_P2" )
      Contact( "bitH_Aut_Man_P2" )
   END_RUNG wire#w2
   RUNG wire#powerrail
      Contact( "IsReady_P4" )
      Contact( "bitH_Aut_Man_P4" )
   END_RUNG wire#w3
   RUNG wire#powerrail
      Contact( "IsReady_P3" )
      Contact( "bitH_Aut_Man_P3" )
   END_RUNG wire#w4
   RUNG wire#powerrail
      Contact( "IsModeAut" )
      Contact( "bitH_Aut_Man_P4" )
   END_RUNG wire#w5
   // the same network as SCL:
   IF NOT "FirstScan" THEN
       "dbSterowanie dołączeniem falownika_P4"(Is_up_Hz := "Is_up_Hz",   // "Sterowanie dołączeniem falownika"
                               Set_HWork_M := "Set_HWork_P4",
                               setPID_Pompy := "setPID_Pompy",
                               IsRunInverter_MA := "IsRunInverter_P1",
                               IsRunNetwork_MA := "IsRunNetwork_P1",
                               IsRunInverter_MB := "IsRunInverter_P2",
                               IsRunNetwork_MB := "IsRunNetwork_P2",
                               IsRunNetwork_MC := "IsRunNetwork_P4",
                               IsRunInverter_MC := "IsRunInverter_P4",
                               IsRunNetwork_MD := "IsRunNetwork_P3",
                               IsRunInverter_MD := "IsRunInverter_P3",
                               FC2_Set_50H := "FC2_Set_50Hz",
                               IsRunInverter1 := "IsRunInverter1",
                               AlwaysTRUE := "AlwaysTRUE",
                               IsReady_MA := "IsReady_P1" AND "bitH_Aut_Man_P1",
                               IsReady_MB := "IsReady_P2" AND "bitH_Aut_Man_P2",
                               IsReady_MC := "IsReady_P4" AND "bitH_Aut_Man_P4",
                               IsReady_MD := "IsReady_P3" AND "bitH_Aut_Man_P3",
                               IsModeAut := "IsModeAut" AND "bitH_Aut_Man_P4",
                               FB9_Set_Motor2 := "FB9_Set_Motor2",
                               FB9_Set_Motor3 := "FB9_Set_Motor3",
                               FB9_Set_Motor4 := "FB9_Set_Motor4",
                               IsReady_Inverter := "IsReady_Inverter",
                               ResWorkInverter_to_MaxTime := "AlwaysFALSE",
                               setCMD_FM := "setCMD_FP4",
                               Timer_OFF_Inverter_M := "dbTimersForDrivers".Timer_OFF_Inverter_P4,
                               Timer_Start_Inver_M := "dbTimersForDrivers".Timer_Start_Inver_P4,
                               Timer_Set50Hz_Off_Inver_M := "dbTimersForDrivers".Timer_Hiteresis_On_Set50Hz_Inver_P4,
                               Mem_Res_setCMD_MC := "dbtags_Sterowanie".SetupControlPompownia.Mem_Res_setCMD_MC_P4,
                               setSUPV_FM => "setSUPV_FP4");
   END_IF;
END_REGION

REGION Network 60: Aktualizacja Trybu PRacy
   // Zabezpieczenie przed zmianami na wypadek anomali
   RUNG wire#powerrail
      I_Contact( "FirstScan" )
      "Korekta Tryb Pracy"()
   END_RUNG
   // the same network as SCL:
   IF NOT "FirstScan" THEN "Korekta Tryb Pracy"(); END_IF;
END_REGION

REGION Network 61: Sterowanie falownikiem
   // Sterowanie załaczaniem falownika
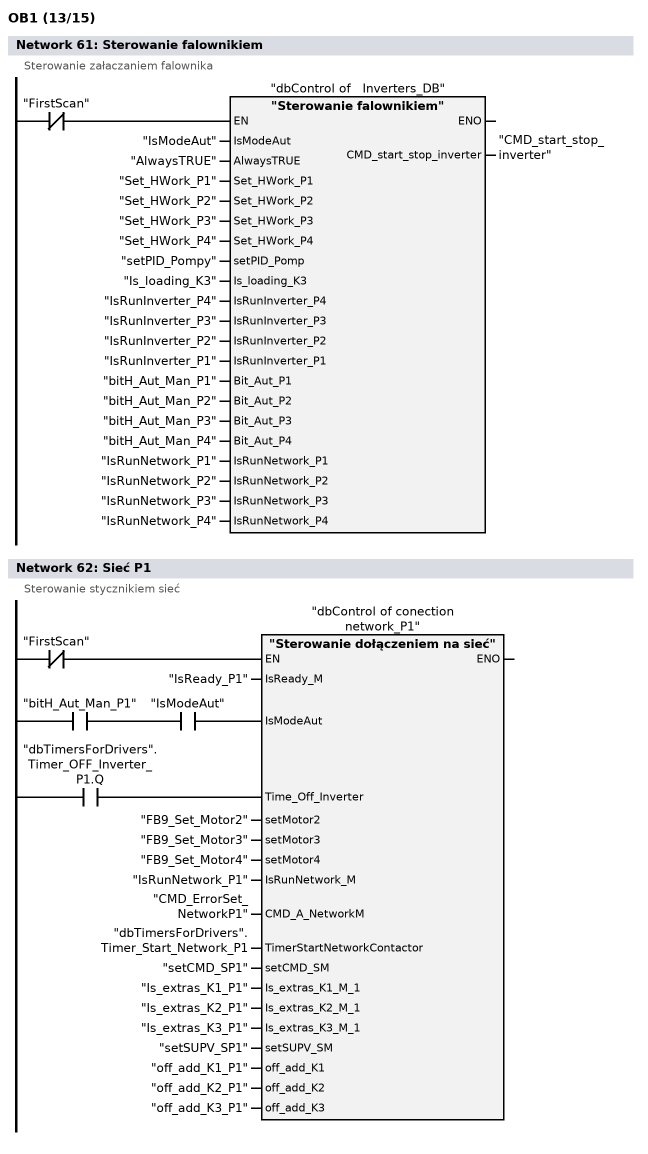
   RUNG wire#powerrail
      I_Contact( "FirstScan" )
      "dbControl of   Inverters_DB"(IsModeAut := "IsModeAut", AlwaysTRUE := "AlwaysTRUE", Set_HWork_P1 := "Set_HWork_P1", Set_HWork_P2 := "Set_HWork_P2", Set_HWork_P3 := "Set_HWork_P3", Set_HWork_P4 := "Set_HWork_P4", setPID_Pomp := "setPID_Pompy", Is_loading_K3 := "Is_loading_K3", IsRunInverter_P4 := "IsRunInverter_P4", IsRunInverter_P3 := "IsRunInverter_P3", IsRunInverter_P2 := "IsRunInverter_P2", IsRunInverter_P1 := "IsRunInverter_P1", Bit_Aut_P1 := "bitH_Aut_Man_P1", Bit_Aut_P2 := "bitH_Aut_Man_P2", Bit_Aut_P3 := "bitH_Aut_Man_P3", Bit_Aut_P4 := "bitH_Aut_Man_P4", IsRunNetwork_P1 := "IsRunNetwork_P1", IsRunNetwork_P2 := "IsRunNetwork_P2", IsRunNetwork_P3 := "IsRunNetwork_P3", IsRunNetwork_P4 := "IsRunNetwork_P4", CMD_start_stop_inverter => "CMD_start_stop_inverter")
   END_RUNG
   // the same network as SCL:
   IF NOT "FirstScan" THEN
       "dbControl of   Inverters_DB"(IsModeAut := "IsModeAut",   // "Sterowanie falownikiem"
                               AlwaysTRUE := "AlwaysTRUE",
                               Set_HWork_P1 := "Set_HWork_P1",
                               Set_HWork_P2 := "Set_HWork_P2",
                               Set_HWork_P3 := "Set_HWork_P3",
                               Set_HWork_P4 := "Set_HWork_P4",
                               setPID_Pomp := "setPID_Pompy",
                               Is_loading_K3 := "Is_loading_K3",
                               IsRunInverter_P4 := "IsRunInverter_P4",
                               IsRunInverter_P3 := "IsRunInverter_P3",
                               IsRunInverter_P2 := "IsRunInverter_P2",
                               IsRunInverter_P1 := "IsRunInverter_P1",
                               Bit_Aut_P1 := "bitH_Aut_Man_P1",
                               Bit_Aut_P2 := "bitH_Aut_Man_P2",
                               Bit_Aut_P3 := "bitH_Aut_Man_P3",
                               Bit_Aut_P4 := "bitH_Aut_Man_P4",
                               IsRunNetwork_P1 := "IsRunNetwork_P1",
                               IsRunNetwork_P2 := "IsRunNetwork_P2",
                               IsRunNetwork_P3 := "IsRunNetwork_P3",
                               IsRunNetwork_P4 := "IsRunNetwork_P4",
                               CMD_start_stop_inverter => "CMD_start_stop_inverter");
   END_IF;
END_REGION

REGION Network 62: Sieć P1
   // Sterowanie stycznikiem sieć
   RUNG wire#powerrail
      I_Contact( "FirstScan" )
      "dbControl of conection network_P1"(IsModeAut := wire#w1, Time_Off_Inverter := wire#w2, IsReady_M := "IsReady_P1", setMotor2 := "FB9_Set_Motor2", setMotor3 := "FB9_Set_Motor3", setMotor4 := "FB9_Set_Motor4", IsRunNetwork_M := "IsRunNetwork_P1", CMD_A_NetworkM := "CMD_ErrorSet_NetworkP1", TimerStartNetworkContactor := "dbTimersForDrivers".Timer_Start_Network_P1, setCMD_SM := "setCMD_SP1", Is_extras_K1_M_1 := "Is_extras_K1_P1", Is_extras_K2_M_1 := "Is_extras_K2_P1", Is_extras_K3_M_1 := "Is_extras_K3_P1", setSUPV_SM := "setSUPV_SP1", off_add_K1 := "off_add_K1_P1", off_add_K2 := "off_add_K2_P1", off_add_K3 := "off_add_K3_P1")
   END_RUNG
   RUNG wire#powerrail
      Contact( "bitH_Aut_Man_P1" )
      Contact( "IsModeAut" )
   END_RUNG wire#w1
   RUNG wire#powerrail
      Contact( "dbTimersForDrivers".Timer_OFF_Inverter_P1.Q )
   END_RUNG wire#w2
   // the same network as SCL:
   IF NOT "FirstScan" THEN
       "dbControl of conection network_P1"(IsReady_M := "IsReady_P1",   // "Sterowanie dołączeniem na sieć"
                               IsModeAut := "bitH_Aut_Man_P1" AND "IsModeAut",
                               Time_Off_Inverter := "dbTimersForDrivers".Timer_OFF_Inverter_P1.Q,
                               setMotor2 := "FB9_Set_Motor2",
                               setMotor3 := "FB9_Set_Motor3",
                               setMotor4 := "FB9_Set_Motor4",
                               IsRunNetwork_M := "IsRunNetwork_P1",
                               CMD_A_NetworkM := "CMD_ErrorSet_NetworkP1",
                               TimerStartNetworkContactor := "dbTimersForDrivers".Timer_Start_Network_P1,
                               setCMD_SM := "setCMD_SP1",
                               Is_extras_K1_M_1 := "Is_extras_K1_P1",
                               Is_extras_K2_M_1 := "Is_extras_K2_P1",
                               Is_extras_K3_M_1 := "Is_extras_K3_P1",
                               setSUPV_SM := "setSUPV_SP1",
                               off_add_K1 := "off_add_K1_P1",
                               off_add_K2 := "off_add_K2_P1",
                               off_add_K3 := "off_add_K3_P1");
   END_IF;
END_REGION

REGION Network 63: Sieć P2
   // Sterowanie stycznikiem sieć
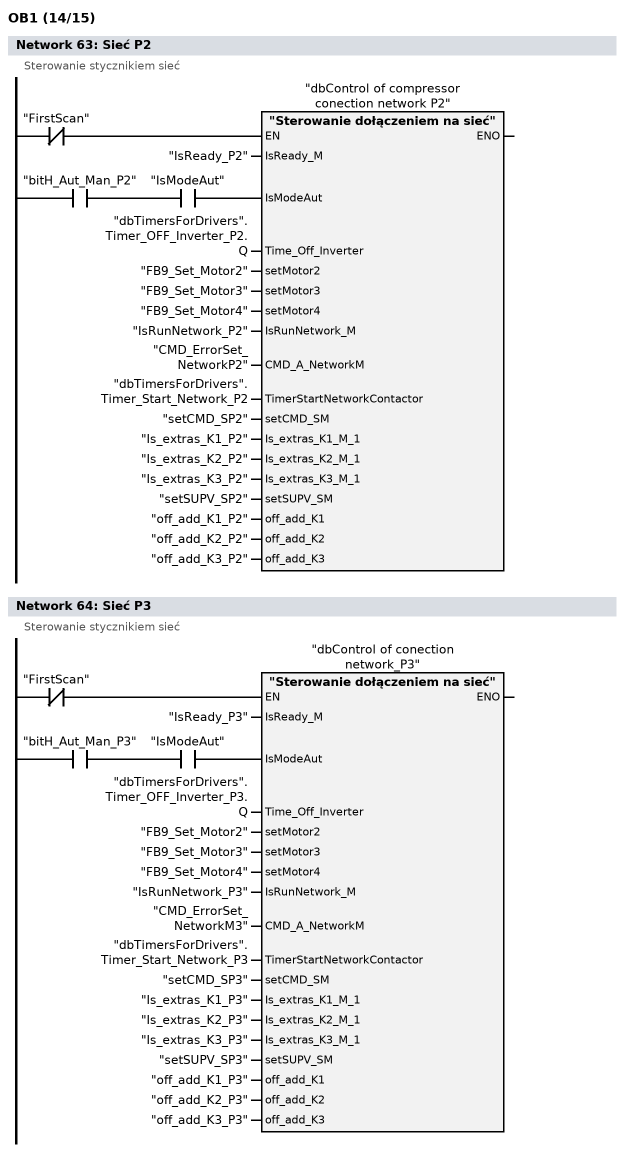
   RUNG wire#powerrail
      I_Contact( "FirstScan" )
      "dbControl of compressor conection network P2"(IsModeAut := wire#w1, IsReady_M := "IsReady_P2", Time_Off_Inverter := "dbTimersForDrivers".Timer_OFF_Inverter_P2.Q, setMotor2 := "FB9_Set_Motor2", setMotor3 := "FB9_Set_Motor3", setMotor4 := "FB9_Set_Motor4", IsRunNetwork_M := "IsRunNetwork_P2", CMD_A_NetworkM := "CMD_ErrorSet_NetworkP2", TimerStartNetworkContactor := "dbTimersForDrivers".Timer_Start_Network_P2, setCMD_SM := "setCMD_SP2", Is_extras_K1_M_1 := "Is_extras_K1_P2", Is_extras_K2_M_1 := "Is_extras_K2_P2", Is_extras_K3_M_1 := "Is_extras_K3_P2", setSUPV_SM := "setSUPV_SP2", off_add_K1 := "off_add_K1_P2", off_add_K2 := "off_add_K2_P2", off_add_K3 := "off_add_K3_P2")
   END_RUNG
   RUNG wire#powerrail
      Contact( "bitH_Aut_Man_P2" )
      Contact( "IsModeAut" )
   END_RUNG wire#w1
   // the same network as SCL:
   IF NOT "FirstScan" THEN
       "dbControl of compressor conection network P2"(IsReady_M := "IsReady_P2",   // "Sterowanie dołączeniem na sieć"
                               IsModeAut := "bitH_Aut_Man_P2" AND "IsModeAut",
                               Time_Off_Inverter := "dbTimersForDrivers".Timer_OFF_Inverter_P2.Q,
                               setMotor2 := "FB9_Set_Motor2",
                               setMotor3 := "FB9_Set_Motor3",
                               setMotor4 := "FB9_Set_Motor4",
                               IsRunNetwork_M := "IsRunNetwork_P2",
                               CMD_A_NetworkM := "CMD_ErrorSet_NetworkP2",
                               TimerStartNetworkContactor := "dbTimersForDrivers".Timer_Start_Network_P2,
                               setCMD_SM := "setCMD_SP2",
                               Is_extras_K1_M_1 := "Is_extras_K1_P2",
                               Is_extras_K2_M_1 := "Is_extras_K2_P2",
                               Is_extras_K3_M_1 := "Is_extras_K3_P2",
                               setSUPV_SM := "setSUPV_SP2",
                               off_add_K1 := "off_add_K1_P2",
                               off_add_K2 := "off_add_K2_P2",
                               off_add_K3 := "off_add_K3_P2");
   END_IF;
END_REGION

REGION Network 64: Sieć P3
   // Sterowanie stycznikiem sieć
   RUNG wire#powerrail
      I_Contact( "FirstScan" )
      "dbControl of conection network_P3"(IsModeAut := wire#w1, IsReady_M := "IsReady_P3", Time_Off_Inverter := "dbTimersForDrivers".Timer_OFF_Inverter_P3.Q, setMotor2 := "FB9_Set_Motor2", setMotor3 := "FB9_Set_Motor3", setMotor4 := "FB9_Set_Motor4", IsRunNetwork_M := "IsRunNetwork_P3", CMD_A_NetworkM := "CMD_ErrorSet_NetworkM3", TimerStartNetworkContactor := "dbTimersForDrivers".Timer_Start_Network_P3, setCMD_SM := "setCMD_SP3", Is_extras_K1_M_1 := "Is_extras_K1_P3", Is_extras_K2_M_1 := "Is_extras_K2_P3", Is_extras_K3_M_1 := "Is_extras_K3_P3", setSUPV_SM := "setSUPV_SP3", off_add_K1 := "off_add_K1_P3", off_add_K2 := "off_add_K2_P3", off_add_K3 := "off_add_K3_P3")
   END_RUNG
   RUNG wire#powerrail
      Contact( "bitH_Aut_Man_P3" )
      Contact( "IsModeAut" )
   END_RUNG wire#w1
   // the same network as SCL:
   IF NOT "FirstScan" THEN
       "dbControl of conection network_P3"(IsReady_M := "IsReady_P3",   // "Sterowanie dołączeniem na sieć"
                               IsModeAut := "bitH_Aut_Man_P3" AND "IsModeAut",
                               Time_Off_Inverter := "dbTimersForDrivers".Timer_OFF_Inverter_P3.Q,
                               setMotor2 := "FB9_Set_Motor2",
                               setMotor3 := "FB9_Set_Motor3",
                               setMotor4 := "FB9_Set_Motor4",
                               IsRunNetwork_M := "IsRunNetwork_P3",
                               CMD_A_NetworkM := "CMD_ErrorSet_NetworkM3",
                               TimerStartNetworkContactor := "dbTimersForDrivers".Timer_Start_Network_P3,
                               setCMD_SM := "setCMD_SP3",
                               Is_extras_K1_M_1 := "Is_extras_K1_P3",
                               Is_extras_K2_M_1 := "Is_extras_K2_P3",
                               Is_extras_K3_M_1 := "Is_extras_K3_P3",
                               setSUPV_SM := "setSUPV_SP3",
                               off_add_K1 := "off_add_K1_P3",
                               off_add_K2 := "off_add_K2_P3",
                               off_add_K3 := "off_add_K3_P3");
   END_IF;
END_REGION

REGION Network 65: Sieć P4
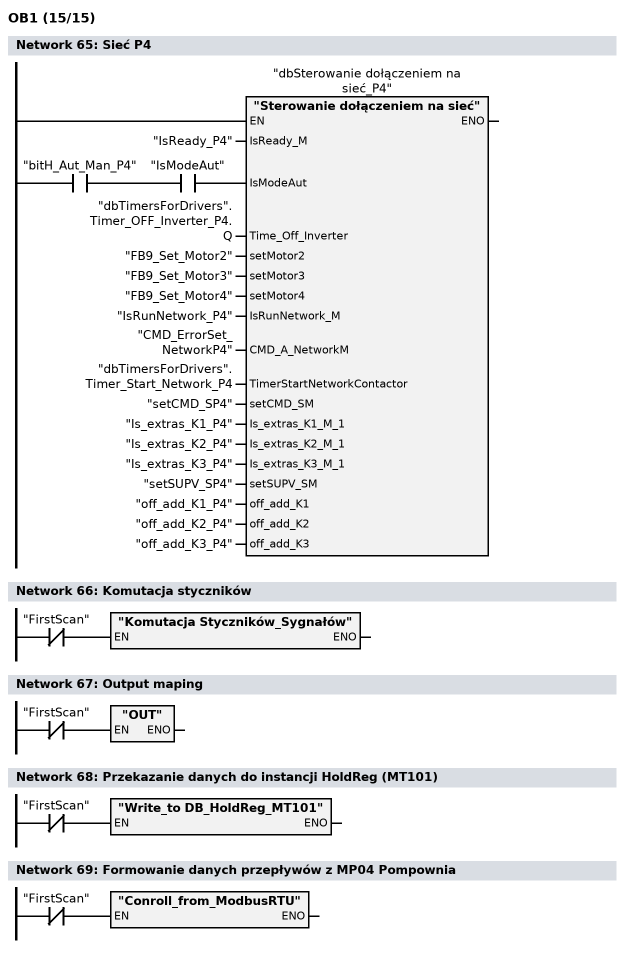
   RUNG wire#powerrail
      "dbSterowanie dołączeniem na sieć_P4"(IsModeAut := wire#w1, IsReady_M := "IsReady_P4", Time_Off_Inverter := "dbTimersForDrivers".Timer_OFF_Inverter_P4.Q, setMotor2 := "FB9_Set_Motor2", setMotor3 := "FB9_Set_Motor3", setMotor4 := "FB9_Set_Motor4", IsRunNetwork_M := "IsRunNetwork_P4", CMD_A_NetworkM := "CMD_ErrorSet_NetworkP4", TimerStartNetworkContactor := "dbTimersForDrivers".Timer_Start_Network_P4, setCMD_SM := "setCMD_SP4", Is_extras_K1_M_1 := "Is_extras_K1_P4", Is_extras_K2_M_1 := "Is_extras_K2_P4", Is_extras_K3_M_1 := "Is_extras_K3_P4", setSUPV_SM := "setSUPV_SP4", off_add_K1 := "off_add_K1_P4", off_add_K2 := "off_add_K2_P4", off_add_K3 := "off_add_K3_P4")
   END_RUNG
   RUNG wire#powerrail
      Contact( "bitH_Aut_Man_P4" )
      Contact( "IsModeAut" )
   END_RUNG wire#w1
   // the same network as SCL:
   "dbSterowanie dołączeniem na sieć_P4"(IsReady_M := "IsReady_P4",   // "Sterowanie dołączeniem na sieć"
                           IsModeAut := "bitH_Aut_Man_P4" AND "IsModeAut",
                           Time_Off_Inverter := "dbTimersForDrivers".Timer_OFF_Inverter_P4.Q,
                           setMotor2 := "FB9_Set_Motor2",
                           setMotor3 := "FB9_Set_Motor3",
                           setMotor4 := "FB9_Set_Motor4",
                           IsRunNetwork_M := "IsRunNetwork_P4",
                           CMD_A_NetworkM := "CMD_ErrorSet_NetworkP4",
                           TimerStartNetworkContactor := "dbTimersForDrivers".Timer_Start_Network_P4,
                           setCMD_SM := "setCMD_SP4",
                           Is_extras_K1_M_1 := "Is_extras_K1_P4",
                           Is_extras_K2_M_1 := "Is_extras_K2_P4",
                           Is_extras_K3_M_1 := "Is_extras_K3_P4",
                           setSUPV_SM := "setSUPV_SP4",
                           off_add_K1 := "off_add_K1_P4",
                           off_add_K2 := "off_add_K2_P4",
                           off_add_K3 := "off_add_K3_P4");
END_REGION

REGION Network 66: Komutacja styczników
   RUNG wire#powerrail
      I_Contact( "FirstScan" )
      "Komutacja Styczników_Sygnałów"()
   END_RUNG
   // the same network as SCL:
   IF NOT "FirstScan" THEN "Komutacja Styczników_Sygnałów"(); END_IF;
END_REGION

REGION Network 67: Output maping
   RUNG wire#powerrail
      I_Contact( "FirstScan" )
      "OUT"()
   END_RUNG
   // the same network as SCL:
   IF NOT "FirstScan" THEN "OUT"(); END_IF;
END_REGION

REGION Network 68: Przekazanie danych do instancji HoldReg (MT101)
   RUNG wire#powerrail
      I_Contact( "FirstScan" )
      "Write_to DB_HoldReg_MT101"()
   END_RUNG
   // the same network as SCL:
   IF NOT "FirstScan" THEN "Write_to DB_HoldReg_MT101"(); END_IF;
END_REGION

REGION Network 69: Formowanie danych przepływów z MP04 Pompownia
   RUNG wire#powerrail
      I_Contact( "FirstScan" )
      "Conroll_from_ModbusRTU"()
   END_RUNG
   // the same network as SCL:
   IF NOT "FirstScan" THEN "Conroll_from_ModbusRTU"(); END_IF;
END_REGION
END_ORGANIZATION_BLOCK
